// TwinCAT 3 PLC project modulx
// ProgramVersion: 3.1.0.8
// libraries:
//   Tc2_Standard, * (Beckhoff Automation GmbH)
//   Tc2_System, * (Beckhoff Automation GmbH)
//   Tc3_Interfaces, * (Beckhoff Automation GmbH)
//   Tc3_Module, * (Beckhoff Automation GmbH)
//   Tc2_MC2,3.3.5.0,Beckhoff Automation GmbH
//   Tc2_TcpIp,3.3.2.0,Beckhoff Automation GmbH
//   Tc2_Utilities,3.3.7.0,Beckhoff Automation GmbH
// project tree:
//   DataTypes/ eMainState.TcDUT, eSubState.TcDUT
//   DUTs/ArrayInterFaceDUT/DUTs/Module Interface/ DUT_MODULE_INTERFACE.TcDUT
//   DUTs/ArrayInterFaceDUT/DUTs/Module Interface/Input/ DUT_MODULE_INTERFACE_INPUT.TcDUT, DUT_SKILL_INPUT.TcDUT
//   DUTs/ArrayInterFaceDUT/DUTs/Module Interface/Output/ DUT_MODULE_INTERFACE_OUTPUT.TcDUT, DUT_SKILL_OUTPUT.TcDUT
//   DUTs/ DUT_SIMULATION.TcDUT
//   DUTs/industrialPhysics/ MNG_APPLICATION_INPUTS_32BIT.TcDUT, MNG_APPLICATION_OUTPUTS_32BIT.TcDUT, MNG_DataArray.TcDUT, MNG_DatagramHeader.TcDUT, MNG_DatagramType.TcDUT, MNG_POSE6.TcDUT, MNG_RawDatagram.TcDUT, MNG_TRAFO.TcDUT, VEC3.TcDUT
//   DUTs/Server DUTs/ DUT_MODE.TcDUT, DUT_PARAMETER_INPUT.TcDUT, DUT_PARAMETER_OUTPUT.TcDUT, DUT_SERVER_MODULE_INTERFACE.TcDUT, DUT_SERVER_MODULE_INTERFACE_INPUT.TcDUT, DUT_SERVER_MODULE_INTERFACE_OUTPUT.TcDUT, DUT_SERVER_PARAMETERINPUTARRAY.TcDUT, DUT_SERVER_PARAMETEROUTPUTARRAY.TcDUT, DUT_SERVER_SKILLINPUTARRAY.TcDUT, DUT_SERVER_SKILLOUTPUTARRAY.TcDUT, DUT_SERVER_SKILL_INPUT.TcDUT, DUT_SERVER_SKILL_OUTPUT.TcDUT, DUT_SERVER_STATEVALUEARRAY.TcDUT, DUT_SIMU_SKILLSTATE.TcDUT, DUT_STATEVALUES.TcDUT
//   GVLs/ GVL.TcGVL, MI5.TcGVL, MNG_GLOBALS.TcGVL, OPCConstants.TcGVL
//   / PlcTask.TcTTO, SimuTask.TcTTO
//   POUs/ FB_FAKE_MODULE.TcPOU, FB_Translate.TcPOU, MAIN.TcPOU
//   POUs/industrialPhysics/ FB_LogFifo.TcPOU, MAIN_simu.TcPOU, MNG_SIMULATION.TcPOU, MNG_UPDATEIOS.TcPOU
// real-time tasks:
//   TASK PlcTask: cycle T#10ms, priority 20, ADS port 350
//   TASK SimuTask: cycle T#10ms, priority 21, ADS port 351
// motion (NC):
//   TASK NC-Task 1 SAF: cycle T#2ms, priority 4, ADS port 501
//   TASK NC-Task 1 SVB: cycle T#10ms, priority 8, ADS port 511

CONFIGURATION modulx
    RESOURCE PLC ON TwinCAT3
        TASK PlcTask(INTERVAL := T#10ms, PRIORITY := 20);
        TASK SimuTask(INTERVAL := T#10ms, PRIORITY := 21);
        PROGRAM MAIN WITH PlcTask : MAIN;
        PROGRAM MAIN_simu WITH SimuTask : MAIN_simu;
    END_RESOURCE
END_CONFIGURATION

// ---- DataTypes/eMainState.TcDUT
TYPE eMainState :
(
	init		:= 0,
	ready		:= 10,
	output		:= 20,
	separation	:= 30,
	refill		:= 40
);
END_TYPE

// ---- DataTypes/eSubState.TcDUT
TYPE eSubState :
(
	step0 := 0,
	step1 := 1,
	step2 := 2,
	step3 := 3,
	step4 := 4,
	step5 := 5,
	step6 := 6,
	step7 := 7,
	step8 := 8,
	step9 := 9,
	step10 := 10,
	step11 := 11,
	step12 := 12,
	step13 := 13,
	step14 := 14,
	step15 := 15
);
END_TYPE

// ---- DUTs/ArrayInterFaceDUT/DUTs/Module Interface/DUT_MODULE_INTERFACE.TcDUT
/// MODULE INTERFACE INPUT AND OUTPUT 
TYPE DUT_MODULE_INTERFACE :
STRUCT
	///Information that the module reads
	Input: DUT_MODULE_INTERFACE_INPUT;
	///Information that the module write
	Output: DUT_MODULE_INTERFACE_OUTPUT;
END_STRUCT
END_TYPE

// ---- DUTs/ArrayInterFaceDUT/DUTs/Module Interface/Input/DUT_MODULE_INTERFACE_INPUT.TcDUT
TYPE DUT_MODULE_INTERFACE_INPUT :
STRUCT
	///Mode to run (init,auto,manual,..)
	Mode: DUT_MODE;
	///check if the modules is alive
	ConnectionTestInput: BOOL;
	///Modules get their position
	PositionInput: LREAL;
	///Update data= TRUE, No updatedata=FALSE
	Watchbit: BOOL;
	///Emergency stop
	EmergencyStop: BOOL;
	///Range of INPUT skills
	SkillInput: ARRAY[0..SkillCnt] OF DUT_SKILL_INPUT;
END_STRUCT
END_TYPE

// ---- DUTs/ArrayInterFaceDUT/DUTs/Module Interface/Input/DUT_SKILL_INPUT.TcDUT
TYPE DUT_SKILL_INPUT :
STRUCT
	///Range of parameters
	ParameterInput: ARRAY[0..ParameterCnt] OF DUT_PARAMETER_INPUT;
	///Start process
	Execute: BOOL;
END_STRUCT
END_TYPE

// ---- DUTs/ArrayInterFaceDUT/DUTs/Module Interface/Output/DUT_MODULE_INTERFACE_OUTPUT.TcDUT
TYPE DUT_MODULE_INTERFACE_OUTPUT :
STRUCT
	///Free to use = TRUE, busy to use =FALSE
	Dummy: BOOL := TRUE;
	///Individual name of the module
	Name: STRING(80);
	///Identification number of module
	ID: UINT;
	///IP address
	IP: STRING(80);
	///Show if the module is in Standby or not
	Idle: BOOL;
	///Show if the module is connected
	Connected: BOOL;
	///Feedback with conection test input
	ConnectionTestOutput: BOOL;
	///Show if the system has error when=TRUE
	Error: BOOL;
	///Identification number of the error
	ErrorID: UINT;
	///Description of the error
	ErrorDescription: STRING(80);
	///Description of the current task
	CurrentTaskDescription: STRING(80);
	///actual position of the modules, calculated by the module itself
	PositionOutput: LREAL;
	///Position of the sensor
	PositionSensor: BOOL;
	///Range of OUTPUT skills
	SkillOutput: ARRAY[0..SkillCnt] OF DUT_SKILL_OUTPUT;
	///Range of state values
	StateValue: ARRAY[0..StateCnt] OF DUT_STATEVALUES;
END_STRUCT
END_TYPE

// ---- DUTs/ArrayInterFaceDUT/DUTs/Module Interface/Output/DUT_SKILL_OUTPUT.TcDUT
TYPE DUT_SKILL_OUTPUT :
STRUCT
	///Free to use = TRUE, busy to use =FALSE
	Dummy: BOOL := TRUE;
	///Identification number of skill
	ID: UINT;
	///indentfication name of skill
	Name: STRING(80);
	///Skill activated
	Activated: BOOL;
	///Ready to do skill
	Ready: BOOL;
	///Skill in process
	Busy: BOOL;
	///Skill finish
	Done: BOOL;
	///Error in system
	Error: BOOL;
	///Range of parameters
	ParameterOutput: ARRAY[0..ParameterCnt] OF DUT_PARAMETER_OUTPUT;
END_STRUCT
END_TYPE

// ---- DUTs/DUT_SIMULATION.TcDUT
TYPE DUT_SIMULATION :
STRUCT
XPosition0 : LREAL;
XPosition1 : lreal;
XPosition2 : lreal;
XPosition3 : lreal;
XPosition4 : lreal;
XPosition5 : lreal;
XPosition6 : lreal;
XPosition7 : lreal;
XPosition8 : lreal;
XPosition9 : lreal;
XPosition10 :LREAL;

Cocktail			: DUT_SIMU_SKILLSTATE;
Cookie				: DUT_SIMU_SKILLSTATE;
Topping_Beckhoff	: DUT_SIMU_SKILLSTATE;
Topping_Bosch		: DUT_SIMU_SKILLSTATE;

END_STRUCT
END_TYPE

// ---- DUTs/industrialPhysics/MNG_APPLICATION_INPUTS_32BIT.TcDUT

TYPE MNG_APPLICATION_INPUTS_32BIT :
STRUCT
    NumSignals                     : INT     := 1         ;
    init_sensor_module_x_00_IR : BOOL    := 0; (* Physics://physics/Modulel_X/init_sensor_module_x?IR *)
END_STRUCT
END_TYPE

// ---- DUTs/industrialPhysics/MNG_APPLICATION_OUTPUTS_32BIT.TcDUT

TYPE MNG_APPLICATION_OUTPUTS_32BIT :
STRUCT
    NumSignals                     : INT     := 18        ;
    MotorX_00_par1 : BOOL    := 0; (* Physics://physics/Modulel_X/MotorX?par1 *)
    MotorX_00_par2 : BOOL    := 0; (* Physics://physics/Modulel_X/MotorX?par2 *)
    Keksmodul_00_ACT_POS02 : REAL    := 0.0; (* Physics://physics/Keksmodul?KinActual *)
    Toppingmodul_Bosch_00_ACT_POS02 : REAL    := 0.0; (* Physics://physics/Toppingmodul_Bosch?KinActual *)
    Toppingmodul_Beckhoff_00_ACT_POS02 : REAL    := 0.0; (* Physics://physics/Toppingmodul_Beckhoff?KinActual *)
    DosierModul_00_ACT_POS02 : REAL    := 0.0; (* Physics://physics/DosierModul?KinActual *)
    status_00_on102 : BOOL    := 0; (* Physics://physics/Keksmodul/status_plate/status?on1 *)
    status_00_on202 : BOOL    := 0; (* Physics://physics/Keksmodul/status_plate/status?on2 *)
    status_00_on302 : BOOL    := 0; (* Physics://physics/Keksmodul/status_plate/status?on3 *)
    status_00_on103 : BOOL    := 0; (* /physics/Toppingmodul_Bosch/status_plate/status?on1 *)
    status_00_on203 : BOOL    := 0; (* /physics/Toppingmodul_Bosch/status_plate/status?on2 *)
    status_00_on303 : BOOL    := 0; (* /physics/Toppingmodul_Bosch/status_plate/status?on3 *)
    status_00_on104 : BOOL    := 0; (* ysics/Toppingmodul_Beckhoff/status_plate/status?on1 *)
    status_00_on204 : BOOL    := 0; (* ysics/Toppingmodul_Beckhoff/status_plate/status?on2 *)
    status_00_on304 : BOOL    := 0; (* ysics/Toppingmodul_Beckhoff/status_plate/status?on3 *)
    status_00_on105 : BOOL    := 0; (* ysics://physics/DosierModul/status_plate/status?on1 *)
    status_00_on205 : BOOL    := 0; (* ysics://physics/DosierModul/status_plate/status?on2 *)
    status_00_on305 : BOOL    := 0; (* ysics://physics/DosierModul/status_plate/status?on3 *)
END_STRUCT
END_TYPE

// ---- DUTs/industrialPhysics/MNG_DataArray.TcDUT
TYPE MNG_DataArray : ARRAY[1..MNG_BUFFER_SIZE] OF DWORD; (* user data of max. length *)
END_TYPE

// ---- DUTs/industrialPhysics/MNG_DatagramHeader.TcDUT
TYPE MNG_DatagramHeader :(* datagram header (4 byte aligned) *)
STRUCT
	(* Time when datagram has been created *)
	Counter 	: DWORD;
	(* Time when datagram has been sent *)
	SentTime 		: DWORD;
	(* Type of the datagram *)
	DatagramType 	: DWORD := MNG_UnknownDatagram;
	(* Byte count in the payload *)
	ByteCount 		: DWORD := 0;
END_STRUCT
END_TYPE

// ---- DUTs/industrialPhysics/MNG_DatagramType.TcDUT
TYPE MNG_DatagramType :
(
	(*Dead man datagram signalizing peer is alive *)
	MNG_DeadManDatagram := 0,
	(*Time tick synchonisation *)
	MNG_TimeTick,
	(*Time tick synchonisation *)
	MNG_TimeTickRequest,
	(*Initialization of the connection *)
	MNG_InitConnection,
	(*Reset simulation *)
	MNG_ResetSimulation,
	(*Rewind simulation *)
	MNG_RewindSimulation,
	(*Start simulation *)
	MNG_StartSimulation,
	(*Stop simulation *)
	MNG_StopSimulation,
	(*IO Config datagram *)
	MNG_IOConfig,
	(*Complete Raw IO Image *)
	MNG_RawIOImage,
	(*Complete Raw 32 Bit IO Image *)
	MNG_Raw32BitImage,
	(*Delta IO, only ios that have changed *)
	(* IODelta, *)
	(*Text datagram *)
	MNG_TextDatagram,
	(*Unknown Datagram (future updates of peer, not supported by this side) *)
	MNG_UnknownDatagram
);
END_TYPE

// ---- DUTs/industrialPhysics/MNG_POSE6.TcDUT
TYPE MNG_POSE6 :(* position and orientation as an euler based pose *)
STRUCT
	x, y, z, a, b, c : REAL;
END_STRUCT
END_TYPE

// ---- DUTs/industrialPhysics/MNG_RawDatagram.TcDUT
TYPE MNG_RawDatagram :(* binary TCP/IP datagram (4 byte aligned) *)
STRUCT
	Header	:  MNG_DatagramHeader;(* datagram header *)
	Payload	:  MNG_DataARRAY;
END_STRUCT
END_TYPE

// ---- DUTs/industrialPhysics/MNG_TRAFO.TcDUT
TYPE MNG_TRAFO :(* position and orientation as a 4x4 matrix *)
STRUCT
	baseX : VEC3; 
	fill0 : REAL;
	baseY : VEC3; 
	fill1 : REAL;
	baseZ : VEC3; 
	fill2 : REAL;
	origin : VEC3;
	fill3 : REAL;
END_STRUCT
END_TYPE

// ---- DUTs/industrialPhysics/VEC3.TcDUT
TYPE VEC3 :(* 3d position *)
STRUCT
	x, y, z : REAL;
END_STRUCT
END_TYPE

// ---- DUTs/Server DUTs/DUT_MODE.TcDUT
/// MODE to run (inside of MODULE_INTERFACE_INPUT)
TYPE DUT_MODE :
(
	///Initialitzation number mode
	Init := 0,
	///Automatic number mode
	Auto := 1,
	///Manual number mode
	Manual := 2,
	Reset := 3
);
END_TYPE

// ---- DUTs/Server DUTs/DUT_PARAMETER_INPUT.TcDUT
TYPE DUT_PARAMETER_INPUT :
STRUCT
	///Value of the parameter 
	Value: LREAL;
	///Possibility to a string value depending on the parameter
	StringValue: STRING(80);
END_STRUCT
END_TYPE

// ---- DUTs/Server DUTs/DUT_PARAMETER_OUTPUT.TcDUT
TYPE DUT_PARAMETER_OUTPUT :
STRUCT
	///Free to use = TRUE, busy to use =FALSE
	Dummy: BOOL := TRUE;
	///ID of the parameter
	ID: UINT;
	///Name of the parameter
	Name: STRING(80);
	///Unit of the parameter
	Unit: STRING(80);
	///Optional parameter
	Required: BOOL;
	///Default parameter to work
	Default: LREAL;
	///Minimum value of the parameter
	MinValue: LREAL;
	///Maximum value of the parameter
	MaxValue: LREAL;
END_STRUCT
END_TYPE

// ---- DUTs/Server DUTs/DUT_SERVER_MODULE_INTERFACE.TcDUT
/// MODULE INTERFACE INPUT AND OUTPUT 
TYPE DUT_SERVER_MODULE_INTERFACE :
STRUCT
	///Information that the module reads
	Input: DUT_SERVER_MODULE_INTERFACE_INPUT;
	///Information that the module write
	Output: DUT_SERVER_MODULE_INTERFACE_OUTPUT;
END_STRUCT
END_TYPE

// ---- DUTs/Server DUTs/DUT_SERVER_MODULE_INTERFACE_INPUT.TcDUT
TYPE DUT_SERVER_MODULE_INTERFACE_INPUT :
STRUCT
	///Mode to run (init,auto,manual,..)
	Mode: INT;//DUT_MODE;
	///check if the modules is alive
	ConnectionTestInput: BOOL;
	///Modules get their position
	PositionInput: LREAL;
	///Update data= TRUE, No updatedata=FALSE
	Watchbit: BOOL;
	///Emergency stop
	EmergencyStop: BOOL;
	///Range of INPUT skills
	SkillInput: DUT_SERVER_SKILLINPUTARRAY;
END_STRUCT
END_TYPE

// ---- DUTs/Server DUTs/DUT_SERVER_MODULE_INTERFACE_OUTPUT.TcDUT
TYPE DUT_SERVER_MODULE_INTERFACE_OUTPUT :
STRUCT
	///Free to use = TRUE, busy to use =FALSE
	Dummy: BOOL := TRUE;
	///Individual name of the module
	Name: STRING(80);
	///Identification number of module
	ID: UINT;
	///IP address
	IP: STRING(80);
	///Show if the module is in Standby or not
	Idle: BOOL;
	///Show if the module is connected
	Connected: BOOL;
	///Feedback with conection test input
	ConnectionTestOutput: BOOL;
	///Show if the system has error when=TRUE
	Error: BOOL;
	///Identification number of the error
	ErrorID: UINT;
	///Description of the error
	ErrorDescription: STRING(80);
	///Description of the current task
	CurrentTaskDescription: STRING(80);
	///Position of the output
	PositionOutput: LREAL;
	/// Bool value of the Sensor
	PositionSensor: BOOL;
	///Range of OUTPUT skills
	SkillOutput: DUT_SERVER_SKILLOUTPUTARRAY;
	///Range of state values
	StateValue: DUT_SERVER_STATEVALUEARRAY;
END_STRUCT
END_TYPE

// ---- DUTs/Server DUTs/DUT_SERVER_PARAMETERINPUTARRAY.TcDUT
TYPE DUT_SERVER_PARAMETERINPUTARRAY :
STRUCT
	ParameterInput0: DUT_PARAMETER_INPUT;
	ParameterInput1: DUT_PARAMETER_INPUT;
	ParameterInput2: DUT_PARAMETER_INPUT;
	ParameterInput3: DUT_PARAMETER_INPUT;
	ParameterInput4: DUT_PARAMETER_INPUT;
	ParameterInput5: DUT_PARAMETER_INPUT;
END_STRUCT
END_TYPE

// ---- DUTs/Server DUTs/DUT_SERVER_PARAMETEROUTPUTARRAY.TcDUT
TYPE DUT_SERVER_PARAMETEROUTPUTARRAY :
STRUCT
	ParameterOutput0: DUT_PARAMETER_OUTPUT;
	ParameterOutput1: DUT_PARAMETER_OUTPUT;
	ParameterOutput2: DUT_PARAMETER_OUTPUT;
	ParameterOutput3: DUT_PARAMETER_OUTPUT;
	ParameterOutput4: DUT_PARAMETER_OUTPUT;
	ParameterOutput5: DUT_PARAMETER_OUTPUT;
END_STRUCT
END_TYPE

// ---- DUTs/Server DUTs/DUT_SERVER_SKILLINPUTARRAY.TcDUT
TYPE DUT_SERVER_SKILLINPUTARRAY :
STRUCT
	SkillInput0: DUT_SERVER_SKILL_INPUT;
	SkillInput1: DUT_SERVER_SKILL_INPUT;
	SkillInput2: DUT_SERVER_SKILL_INPUT;
	SkillInput3: DUT_SERVER_SKILL_INPUT;
	SkillInput4: DUT_SERVER_SKILL_INPUT;
	SkillInput5: DUT_SERVER_SKILL_INPUT;
	SkillInput6: DUT_SERVER_SKILL_INPUT;
	SkillInput7: DUT_SERVER_SKILL_INPUT;
	SkillInput8: DUT_SERVER_SKILL_INPUT;
	SkillInput9: DUT_SERVER_SKILL_INPUT;
	SkillInput10: DUT_SERVER_SKILL_INPUT;
	SkillInput11: DUT_SERVER_SKILL_INPUT;
	SkillInput12: DUT_SERVER_SKILL_INPUT;
	SkillInput13: DUT_SERVER_SKILL_INPUT;
	SkillInput14: DUT_SERVER_SKILL_INPUT;
	SkillInput15: DUT_SERVER_SKILL_INPUT;
END_STRUCT
END_TYPE

// ---- DUTs/Server DUTs/DUT_SERVER_SKILLOUTPUTARRAY.TcDUT
TYPE DUT_SERVER_SKILLOUTPUTARRAY :
STRUCT
	SkillOutput0: DUT_SERVER_SKILL_OUTPUT;
	SkillOutput1: DUT_SERVER_SKILL_OUTPUT;
	SkillOutput2: DUT_SERVER_SKILL_OUTPUT;
	SkillOutput3: DUT_SERVER_SKILL_OUTPUT;
	SkillOutput4: DUT_SERVER_SKILL_OUTPUT;
	SkillOutput5: DUT_SERVER_SKILL_OUTPUT;
	SkillOutput6: DUT_SERVER_SKILL_OUTPUT;
	SkillOutput7: DUT_SERVER_SKILL_OUTPUT;
	SkillOutput8: DUT_SERVER_SKILL_OUTPUT;
	SkillOutput9: DUT_SERVER_SKILL_OUTPUT;
	SkillOutput10: DUT_SERVER_SKILL_OUTPUT;
	SkillOutput11: DUT_SERVER_SKILL_OUTPUT;
	SkillOutput12: DUT_SERVER_SKILL_OUTPUT;
	SkillOutput13: DUT_SERVER_SKILL_OUTPUT;
	SkillOutput14: DUT_SERVER_SKILL_OUTPUT;
	SkillOutput15: DUT_SERVER_SKILL_OUTPUT;
END_STRUCT
END_TYPE

// ---- DUTs/Server DUTs/DUT_SERVER_SKILL_INPUT.TcDUT
TYPE DUT_SERVER_SKILL_INPUT :
STRUCT
	///Range of parameters
	ParameterInput: DUT_SERVER_PARAMETERINPUTARRAY;
	///Start process
	Execute: BOOL;
END_STRUCT
END_TYPE

// ---- DUTs/Server DUTs/DUT_SERVER_SKILL_OUTPUT.TcDUT
TYPE DUT_SERVER_SKILL_OUTPUT :
STRUCT
	///Free to use = TRUE, busy to use =FALSE
	Dummy: BOOL := TRUE;
	///Identification number of skill
	ID: UINT;
	///indentfication name of skill
	Name: STRING(80);
	///Skill activated
	Activated: BOOL;
	///Ready to do skill
	Ready: BOOL;
	///Skill in process
	Busy: BOOL;
	///Skill finish
	Done: BOOL;
	///Error in system
	Error: BOOL;
	///Range of parameters
	ParameterOutput: DUT_SERVER_PARAMETEROUTPUTARRAY;
END_STRUCT
END_TYPE

// ---- DUTs/Server DUTs/DUT_SERVER_STATEVALUEARRAY.TcDUT
TYPE DUT_SERVER_STATEVALUEARRAY :
STRUCT
	StateValue0: DUT_STATEVALUES;
	StateValue1: DUT_STATEVALUES;
	StateValue2: DUT_STATEVALUES;
	StateValue3: DUT_STATEVALUES;
	StateValue4: DUT_STATEVALUES;
	StateValue5: DUT_STATEVALUES;
	StateValue6: DUT_STATEVALUES;
	StateValue7: DUT_STATEVALUES;
	StateValue8: DUT_STATEVALUES;
	StateValue9: DUT_STATEVALUES;
	StateValue10: DUT_STATEVALUES;
END_STRUCT
END_TYPE

// ---- DUTs/Server DUTs/DUT_SIMU_SKILLSTATE.TcDUT
TYPE DUT_SIMU_SKILLSTATE :
STRUCT
	
Ready 	:BOOL;
Busy	:BOOL;
Error	:BOOL;

END_STRUCT
END_TYPE

// ---- DUTs/Server DUTs/DUT_STATEVALUES.TcDUT
TYPE DUT_STATEVALUES :
STRUCT
	///Free to use = TRUE, busy to use =FALSE
	Dummy: BOOL := TRUE;
	///Value of the State
	Value: LREAL;
	///Name of the state
	Name: STRING(80);
	///Description of the state
	Description: STRING(80);
	///Unit of the state ()
	Unit: STRING(80);
END_STRUCT
END_TYPE

// ---- GVLs/GVL.TcGVL
VAR_GLOBAL
	pi : REAL := 3.14159;
																
	//<<Input Variables>>//
	iOrder 			AT%I*	: BOOL; 				// is there a order to separate cookies? --> from database
	iDiskAtStorage 	AT%I*	: BOOL; 				// is the gap of the disk at the storage? --> from hall sensor
	iDiskAtRamp 	AT%I*	: BOOL;					// is the gap of the disk at the ramp? --> from hall sensor
	iCookieInOutput	AT%I*	: BOOL;					// is the cookie in the ouput (on the clamp)? --> from light barrier sensor
	iStorageLevel 	AT%I*	: INT;					// number of remaining cookies in the storage --> from distance sensor
	iClearence		AT%I*	: BOOL;					// did the user clear the refilling/maintenance process --> from HMI
	
	//<<Output Variables>>//
	oTurnDiskLeft	AT%Q*	: BOOL := FALSE;		// turn disk anti-clockwise/left 
										 			//@TODO: later as a function with choosable fastVel/acceleration/...
	oTurnDiskRight	AT%Q*	: BOOL := FALSE;		// turn disk anti-clockwise/left 
										 			//@TODO: later as a function with choosable fastVel/acceleration/...							
	//oStorageEmpty	AT%Q*	: BOOL := FALSE;		// ???? message to HMI about cookie storage
	oHMIMessage		AT%Q*	: STRING :='';			//message to HMI depending on current state
	
	//<<Internal Variables>>//
	mainState 				: eMainState		:= eMainState.init;
	subState				: eSubState 		:= eSubState.step0;	
	
	axis	 				: AXIS_REF;
	fastVel					: INT	:= 40;
	slowVel					: INT	:= 20;
	
	
	
	
	//<<For Visualization>>//
	init_					: BOOL := FALSE;
	ready_					: BOOL := FALSE;
	output_					: BOOL := FALSE;
	separation_				: BOOL := FALSE;
	refill_					: BOOL := FALSE;
	
	offset					: LREAL;
	infinitsimu				: BOOL;
	infinitsimu2			: BOOL;	
	sensorPosition			: LREAL;
	
	init_sensor_x			: BOOL;
	lamp1				: BOOL;
	lamp2				: BOOL;	
END_VAR

// ---- GVLs/MI5.TcGVL
VAR_GLOBAL
	//<<OPC-UA Module Interface>>//
	{attribute 'OPC.UA.DA' := '1'}
	Module1202 : DUT_SERVER_MODULE_INTERFACE;
	{attribute 'OPC.UA.DA' := '1'}
	Module2501 : DUT_SERVER_MODULE_INTERFACE;
	{attribute 'OPC.UA.DA' := '1'}
	Module2601 : DUT_SERVER_MODULE_INTERFACE;
	{attribute 'OPC.UA.DA' := '1'}
	Simulation: DUT_SIMULATION;
	{attribute 'OPC.UA.DA' := '1'}	
	ResetProcessTool 	: BOOL;
	
	// INTERN MODULE INTERFACE
	InternalModule	: DUT_MODULE_INTERFACE;
END_VAR

// ---- GVLs/MNG_GLOBALS.TcGVL

VAR_GLOBAL CONSTANT
	PLCPRJ_MAX_CONNECTIONS					: UDINT 	:= 5;   (* Max. number of server<->client connections *)
	PLCPRJ_SERVER_RESPONSE_TIMEOUT			: TIME 	:= T#10s;
	PLCPRJ_CLIENT_SEND_CYCLE_TIME			: TIME 	:= T#1ms;

	PLCPRJ_RECEIVER_POLLING_CYCLE_TIME		: TIME 	:= T#1ms;
	PLCPRJ_BUFFER_SIZE						: UDINT	:= 10000;   (* Max. internal fifo/receiver buffer size *)

	(* Some project specific error codes *)
	PLCPRJ_ERROR_RECEIVE_BUFFER_OVERFLOW	: UDINT := 16#8101; (* receive fifo/buffer overflow*)
	PLCPRJ_ERROR_SEND_BUFFER_OVERFLOW		: UDINT := 16#8102;	(* send fifo/buffer overflow *)
	PLCPRJ_ERROR_RESPONSE_TIMEOUT			: UDINT := 16#8103;	(* receive timeout error *)
	
	

	PLCPRJ_ERROR_INVALID_FRAME_FORMAT		: UDINT := 16#8104;	(* invalid frame format/data *)
	PLCPRJ_ERROR_INVALID_IO_FORMAT_RECEIVED : UDINT := 16#8105;	(* invalid io format/data *)
	PLCPRJ_ERROR_INTERNAL					: UDINT := 16#8105; (* internal error *)
	PLCPRJ_ERROR_RX_DATA_INCONSISTENT		: UDINT := 16#8106; (* rx data inconsistent *)
	
	PLCPRJ_ERROR_RECEIVE_TIMEOUT			: UDINT := 16#8107;
	PLCPRJ_ERROR_SENDFIFO_OVERFLOW			: UDINT := 16#8108; (* send fifo overflow error *)
	PLCPRJ_ERROR_RECFIFO_OVERFLOW			: UDINT := 16#8109; (* receive fifo overflow error *)
	
    MNG_BUFFER_SIZE						: DWORD := 32768;   (* Bytes: 131072; Max 128 KB of datagram payload data*)
	MNG_DatagramsFIFO_Size					: DWORD := 10;      (* Max 10 datagrams buffered before loss occurs *)
	MNG_EmptyDatagramHeader					: MNG_DatagramHeader;
	MNG_Application_NumInputs				: DWORD := 4;
	MNG_Application_NumOutputs				: DWORD := 4;

        (* PI should be defined by the system *)
        (* PI      : LREAL := 3.1415926535897932384626433832795; *)
        DEG2RAD : LREAL := 0.017453292519943295769236907684886;
        RAD2DEG : LREAL := 57.295779513082320876798154814105;
END_VAR

VAR_GLOBAL
        MNG_TIMESTAMP                                           : LREAL := 0;
END_VAR

// ---- GVLs/OPCConstants.TcGVL
VAR_GLOBAL CONSTANT
	///Maximum number of skillparameters
	ParameterCnt: INT := 5;
	///Maximum number of skills per Module
	SkillCnt: INT := 15;
	///Maximum number of Statevalues of one Module
	StateCnt: INT := 10;
	///Maximum number of modules
	ModuleCnt: INT := 10;
	///Maximum number of Tasks in Production List
	TaskCnt: INT := 30;
	///Maximum number  of offered recipes
	OfferCnt: INT := 5;
	///Maximum number of Orders in Queue
	OrderCnt: INT := 5;
	///Number of user set parameters per recipe
	UserParameterCnt: INT := 5;
	///Number of skills per task
	TaskSkillCnt: INT := 50;
END_VAR

// ---- POUs/MAIN.TcPOU
PROGRAM MAIN
VAR


	
	fbTranslate		: FB_TRANSLATE;
	fbFakeModule	: FB_FAKE_MODULE;
	fbi_Timer: TOF;
END_VAR


//für dieses modul muss Module1102 (ausgang von fbTranslate) noch auf den richtigen modulausgang geändert werden und in den GVLs eine Variable vom Typ DUT_Module_Interface (mit arrays) und dem namen InternalModule hinzugefügt werden
// FAKE MODUL:	
fbFakeModule.SKILLID[0] := 1337;

fbFakeModule(INPUT:=InternalModule.Input, OUTPUT => InternalModule.Output,  Execute := TRUE );
fbTranslate(ArrayModule := InternalModule, ServerModule := Module1202);
fbi_Timer();

// sensorhigh delay erzeugen/verlängern
IF GVL.init_sensor_x THEN
	Module1202.Output.PositionSensor := TRUE;
	
	fbi_Timer(IN := TRUE,PT := T#400MS);
	fbi_Timer(IN := FALSE,PT := T#400MS);	
ELSE
	Module1202.Output.PositionSensor := fbi_Timer.Q;
END_IF

Module2501.Output.PositionOutput := 1345.0;
Module2601.Output.PositionOutput := 165.0;

END_PROGRAM

// ---- POUs/FB_Translate.TcPOU
FUNCTION_BLOCK FB_Translate
VAR_INPUT
	execute : BOOL := TRUE;
END_VAR
VAR_OUTPUT
END_VAR
VAR

 
END_VAR
VAR_IN_OUT
	ArrayModule	: DUT_MODULE_INTERFACE;
	ServerModule: DUT_SERVER_MODULE_INTERFACE;
END_VAR

IF execute THEN
	ArrayModule.Input.Mode := ServerModule.Input.Mode;
ArrayModule.Input.ConnectionTestInput := ServerModule.Input.ConnectionTestInput;
ArrayModule.Input.PositionInput := ServerModule.Input.PositionInput;
ArrayModule.Input.Watchbit := ServerModule.Input.Watchbit;
ArrayModule.Input.EmergencyStop := ServerModule.Input.EmergencyStop;
ServerModule.Output.Dummy := ArrayModule.Output.Dummy;
ServerModule.Output.Name := ArrayModule.Output.Name;
ServerModule.Output.ID := ArrayModule.Output.ID;
ServerModule.Output.IP := ArrayModule.Output.IP;
ServerModule.Output.Idle := ArrayModule.Output.Idle;
ServerModule.Output.Connected := ArrayModule.Output.Connected;
ServerModule.Output.Error := ArrayModule.Output.Error;
ServerModule.Output.ErrorID := ArrayModule.Output.ErrorID;
ServerModule.Output.ErrorDescription := ArrayModule.Output.ErrorDescription;
ServerModule.Output.CurrentTaskDescription := ArrayModule.Output.CurrentTaskDescription;
ServerModule.Output.PositionSensor := ArrayModule.Output.PositionSensor;
ServerModule.Output.ConnectionTestOutput := ArrayModule.Output.ConnectionTestOutput;
ServerModule.Output.PositionOutput := ArrayModule.Output.PositionOutput;
ArrayModule.Input.SkillInput[0].Execute := ServerModule.Input.SkillInput.SkillInput0.Execute;
ServerModule.Output.SkillOutput.SkillOutput0.Dummy := ArrayModule.Output.SkillOutput[0].Dummy;
ServerModule.Output.SkillOutput.SkillOutput0.ID := ArrayModule.Output.SkillOutput[0].ID;
ServerModule.Output.SkillOutput.SkillOutput0.Name := ArrayModule.Output.SkillOutput[0].Name;
ServerModule.Output.SkillOutput.SkillOutput0.Activated := ArrayModule.Output.SkillOutput[0].Activated;
ServerModule.Output.SkillOutput.SkillOutput0.Ready := ArrayModule.Output.SkillOutput[0].Ready;
ServerModule.Output.SkillOutput.SkillOutput0.Busy := ArrayModule.Output.SkillOutput[0].Busy;
ServerModule.Output.SkillOutput.SkillOutput0.Done := ArrayModule.Output.SkillOutput[0].Done;
ServerModule.Output.SkillOutput.SkillOutput0.Error := ArrayModule.Output.SkillOutput[0].Error;
ServerModule.Output.Statevalue.Statevalue0 := ArrayModule.Output.Statevalue[0];
ServerModule.Output.Statevalue.Statevalue1 := ArrayModule.Output.Statevalue[1];
ServerModule.Output.Statevalue.Statevalue2 := ArrayModule.Output.Statevalue[2];
ServerModule.Output.Statevalue.Statevalue3 := ArrayModule.Output.Statevalue[3];
ServerModule.Output.Statevalue.Statevalue4 := ArrayModule.Output.Statevalue[4];
ServerModule.Output.Statevalue.Statevalue5 := ArrayModule.Output.Statevalue[5];
ServerModule.Output.Statevalue.Statevalue6 := ArrayModule.Output.Statevalue[6];
ServerModule.Output.Statevalue.Statevalue7 := ArrayModule.Output.Statevalue[7];
ServerModule.Output.Statevalue.Statevalue8 := ArrayModule.Output.Statevalue[8];
ServerModule.Output.Statevalue.Statevalue9 := ArrayModule.Output.Statevalue[9];
ServerModule.Output.Statevalue.Statevalue10 := ArrayModule.Output.Statevalue[10];
ArrayModule.Input.SkillInput[0].ParameterInput[0] := ServerModule.Input.SkillInput.SkillInput0.ParameterInput.ParameterInput0;
ServerModule.Output.SkillOutput.SkillOutput0.ParameterOutput.ParameterOutput0 := ArrayModule.Output.SkillOutput[0].ParameterOutput[0];
ArrayModule.Input.SkillInput[0].ParameterInput[1] := ServerModule.Input.SkillInput.SkillInput0.ParameterInput.ParameterInput1;
ServerModule.Output.SkillOutput.SkillOutput0.ParameterOutput.ParameterOutput1 := ArrayModule.Output.SkillOutput[0].ParameterOutput[1];
ArrayModule.Input.SkillInput[0].ParameterInput[2] := ServerModule.Input.SkillInput.SkillInput0.ParameterInput.ParameterInput2;
ServerModule.Output.SkillOutput.SkillOutput0.ParameterOutput.ParameterOutput2 := ArrayModule.Output.SkillOutput[0].ParameterOutput[2];
ArrayModule.Input.SkillInput[0].ParameterInput[3] := ServerModule.Input.SkillInput.SkillInput0.ParameterInput.ParameterInput3;
ServerModule.Output.SkillOutput.SkillOutput0.ParameterOutput.ParameterOutput3 := ArrayModule.Output.SkillOutput[0].ParameterOutput[3];
ArrayModule.Input.SkillInput[0].ParameterInput[4] := ServerModule.Input.SkillInput.SkillInput0.ParameterInput.ParameterInput4;
ServerModule.Output.SkillOutput.SkillOutput0.ParameterOutput.ParameterOutput4 := ArrayModule.Output.SkillOutput[0].ParameterOutput[4];
ArrayModule.Input.SkillInput[0].ParameterInput[5] := ServerModule.Input.SkillInput.SkillInput0.ParameterInput.ParameterInput5;
ServerModule.Output.SkillOutput.SkillOutput0.ParameterOutput.ParameterOutput5 := ArrayModule.Output.SkillOutput[0].ParameterOutput[5];
ArrayModule.Input.SkillInput[1].Execute := ServerModule.Input.SkillInput.SkillInput1.Execute;
ServerModule.Output.SkillOutput.SkillOutput1.Dummy := ArrayModule.Output.SkillOutput[1].Dummy;
ServerModule.Output.SkillOutput.SkillOutput1.ID := ArrayModule.Output.SkillOutput[1].ID;
ServerModule.Output.SkillOutput.SkillOutput1.Name := ArrayModule.Output.SkillOutput[1].Name;
ServerModule.Output.SkillOutput.SkillOutput1.Activated := ArrayModule.Output.SkillOutput[1].Activated;
ServerModule.Output.SkillOutput.SkillOutput1.Ready := ArrayModule.Output.SkillOutput[1].Ready;
ServerModule.Output.SkillOutput.SkillOutput1.Busy := ArrayModule.Output.SkillOutput[1].Busy;
ServerModule.Output.SkillOutput.SkillOutput1.Done := ArrayModule.Output.SkillOutput[1].Done;
ServerModule.Output.SkillOutput.SkillOutput1.Error := ArrayModule.Output.SkillOutput[1].Error;
ServerModule.Output.Statevalue.Statevalue0 := ArrayModule.Output.Statevalue[0];
ServerModule.Output.Statevalue.Statevalue1 := ArrayModule.Output.Statevalue[1];
ServerModule.Output.Statevalue.Statevalue2 := ArrayModule.Output.Statevalue[2];
ServerModule.Output.Statevalue.Statevalue3 := ArrayModule.Output.Statevalue[3];
ServerModule.Output.Statevalue.Statevalue4 := ArrayModule.Output.Statevalue[4];
ServerModule.Output.Statevalue.Statevalue5 := ArrayModule.Output.Statevalue[5];
ServerModule.Output.Statevalue.Statevalue6 := ArrayModule.Output.Statevalue[6];
ServerModule.Output.Statevalue.Statevalue7 := ArrayModule.Output.Statevalue[7];
ServerModule.Output.Statevalue.Statevalue8 := ArrayModule.Output.Statevalue[8];
ServerModule.Output.Statevalue.Statevalue9 := ArrayModule.Output.Statevalue[9];
ServerModule.Output.Statevalue.Statevalue10 := ArrayModule.Output.Statevalue[10];
ArrayModule.Input.SkillInput[1].ParameterInput[0] := ServerModule.Input.SkillInput.SkillInput1.ParameterInput.ParameterInput0;
ServerModule.Output.SkillOutput.SkillOutput1.ParameterOutput.ParameterOutput0 := ArrayModule.Output.SkillOutput[1].ParameterOutput[0];
ArrayModule.Input.SkillInput[1].ParameterInput[1] := ServerModule.Input.SkillInput.SkillInput1.ParameterInput.ParameterInput1;
ServerModule.Output.SkillOutput.SkillOutput1.ParameterOutput.ParameterOutput1 := ArrayModule.Output.SkillOutput[1].ParameterOutput[1];
ArrayModule.Input.SkillInput[1].ParameterInput[2] := ServerModule.Input.SkillInput.SkillInput1.ParameterInput.ParameterInput2;
ServerModule.Output.SkillOutput.SkillOutput1.ParameterOutput.ParameterOutput2 := ArrayModule.Output.SkillOutput[1].ParameterOutput[2];
ArrayModule.Input.SkillInput[1].ParameterInput[3] := ServerModule.Input.SkillInput.SkillInput1.ParameterInput.ParameterInput3;
ServerModule.Output.SkillOutput.SkillOutput1.ParameterOutput.ParameterOutput3 := ArrayModule.Output.SkillOutput[1].ParameterOutput[3];
ArrayModule.Input.SkillInput[1].ParameterInput[4] := ServerModule.Input.SkillInput.SkillInput1.ParameterInput.ParameterInput4;
ServerModule.Output.SkillOutput.SkillOutput1.ParameterOutput.ParameterOutput4 := ArrayModule.Output.SkillOutput[1].ParameterOutput[4];
ArrayModule.Input.SkillInput[1].ParameterInput[5] := ServerModule.Input.SkillInput.SkillInput1.ParameterInput.ParameterInput5;
ServerModule.Output.SkillOutput.SkillOutput1.ParameterOutput.ParameterOutput5 := ArrayModule.Output.SkillOutput[1].ParameterOutput[5];
ArrayModule.Input.SkillInput[2].Execute := ServerModule.Input.SkillInput.SkillInput2.Execute;
ServerModule.Output.SkillOutput.SkillOutput2.Dummy := ArrayModule.Output.SkillOutput[2].Dummy;
ServerModule.Output.SkillOutput.SkillOutput2.ID := ArrayModule.Output.SkillOutput[2].ID;
ServerModule.Output.SkillOutput.SkillOutput2.Name := ArrayModule.Output.SkillOutput[2].Name;
ServerModule.Output.SkillOutput.SkillOutput2.Activated := ArrayModule.Output.SkillOutput[2].Activated;
ServerModule.Output.SkillOutput.SkillOutput2.Ready := ArrayModule.Output.SkillOutput[2].Ready;
ServerModule.Output.SkillOutput.SkillOutput2.Busy := ArrayModule.Output.SkillOutput[2].Busy;
ServerModule.Output.SkillOutput.SkillOutput2.Done := ArrayModule.Output.SkillOutput[2].Done;
ServerModule.Output.SkillOutput.SkillOutput2.Error := ArrayModule.Output.SkillOutput[2].Error;
ServerModule.Output.Statevalue.Statevalue0 := ArrayModule.Output.Statevalue[0];
ServerModule.Output.Statevalue.Statevalue1 := ArrayModule.Output.Statevalue[1];
ServerModule.Output.Statevalue.Statevalue2 := ArrayModule.Output.Statevalue[2];
ServerModule.Output.Statevalue.Statevalue3 := ArrayModule.Output.Statevalue[3];
ServerModule.Output.Statevalue.Statevalue4 := ArrayModule.Output.Statevalue[4];
ServerModule.Output.Statevalue.Statevalue5 := ArrayModule.Output.Statevalue[5];
ServerModule.Output.Statevalue.Statevalue6 := ArrayModule.Output.Statevalue[6];
ServerModule.Output.Statevalue.Statevalue7 := ArrayModule.Output.Statevalue[7];
ServerModule.Output.Statevalue.Statevalue8 := ArrayModule.Output.Statevalue[8];
ServerModule.Output.Statevalue.Statevalue9 := ArrayModule.Output.Statevalue[9];
ServerModule.Output.Statevalue.Statevalue10 := ArrayModule.Output.Statevalue[10];
ArrayModule.Input.SkillInput[2].ParameterInput[0] := ServerModule.Input.SkillInput.SkillInput2.ParameterInput.ParameterInput0;
ServerModule.Output.SkillOutput.SkillOutput2.ParameterOutput.ParameterOutput0 := ArrayModule.Output.SkillOutput[2].ParameterOutput[0];
ArrayModule.Input.SkillInput[2].ParameterInput[1] := ServerModule.Input.SkillInput.SkillInput2.ParameterInput.ParameterInput1;
ServerModule.Output.SkillOutput.SkillOutput2.ParameterOutput.ParameterOutput1 := ArrayModule.Output.SkillOutput[2].ParameterOutput[1];
ArrayModule.Input.SkillInput[2].ParameterInput[2] := ServerModule.Input.SkillInput.SkillInput2.ParameterInput.ParameterInput2;
ServerModule.Output.SkillOutput.SkillOutput2.ParameterOutput.ParameterOutput2 := ArrayModule.Output.SkillOutput[2].ParameterOutput[2];
ArrayModule.Input.SkillInput[2].ParameterInput[3] := ServerModule.Input.SkillInput.SkillInput2.ParameterInput.ParameterInput3;
ServerModule.Output.SkillOutput.SkillOutput2.ParameterOutput.ParameterOutput3 := ArrayModule.Output.SkillOutput[2].ParameterOutput[3];
ArrayModule.Input.SkillInput[2].ParameterInput[4] := ServerModule.Input.SkillInput.SkillInput2.ParameterInput.ParameterInput4;
ServerModule.Output.SkillOutput.SkillOutput2.ParameterOutput.ParameterOutput4 := ArrayModule.Output.SkillOutput[2].ParameterOutput[4];
ArrayModule.Input.SkillInput[2].ParameterInput[5] := ServerModule.Input.SkillInput.SkillInput2.ParameterInput.ParameterInput5;
ServerModule.Output.SkillOutput.SkillOutput2.ParameterOutput.ParameterOutput5 := ArrayModule.Output.SkillOutput[2].ParameterOutput[5];
ArrayModule.Input.SkillInput[3].Execute := ServerModule.Input.SkillInput.SkillInput3.Execute;
ServerModule.Output.SkillOutput.SkillOutput3.Dummy := ArrayModule.Output.SkillOutput[3].Dummy;
ServerModule.Output.SkillOutput.SkillOutput3.ID := ArrayModule.Output.SkillOutput[3].ID;
ServerModule.Output.SkillOutput.SkillOutput3.Name := ArrayModule.Output.SkillOutput[3].Name;
ServerModule.Output.SkillOutput.SkillOutput3.Activated := ArrayModule.Output.SkillOutput[3].Activated;
ServerModule.Output.SkillOutput.SkillOutput3.Ready := ArrayModule.Output.SkillOutput[3].Ready;
ServerModule.Output.SkillOutput.SkillOutput3.Busy := ArrayModule.Output.SkillOutput[3].Busy;
ServerModule.Output.SkillOutput.SkillOutput3.Done := ArrayModule.Output.SkillOutput[3].Done;
ServerModule.Output.SkillOutput.SkillOutput3.Error := ArrayModule.Output.SkillOutput[3].Error;
ServerModule.Output.Statevalue.Statevalue0 := ArrayModule.Output.Statevalue[0];
ServerModule.Output.Statevalue.Statevalue1 := ArrayModule.Output.Statevalue[1];
ServerModule.Output.Statevalue.Statevalue2 := ArrayModule.Output.Statevalue[2];
ServerModule.Output.Statevalue.Statevalue3 := ArrayModule.Output.Statevalue[3];
ServerModule.Output.Statevalue.Statevalue4 := ArrayModule.Output.Statevalue[4];
ServerModule.Output.Statevalue.Statevalue5 := ArrayModule.Output.Statevalue[5];
ServerModule.Output.Statevalue.Statevalue6 := ArrayModule.Output.Statevalue[6];
ServerModule.Output.Statevalue.Statevalue7 := ArrayModule.Output.Statevalue[7];
ServerModule.Output.Statevalue.Statevalue8 := ArrayModule.Output.Statevalue[8];
ServerModule.Output.Statevalue.Statevalue9 := ArrayModule.Output.Statevalue[9];
ServerModule.Output.Statevalue.Statevalue10 := ArrayModule.Output.Statevalue[10];
ArrayModule.Input.SkillInput[3].ParameterInput[0] := ServerModule.Input.SkillInput.SkillInput3.ParameterInput.ParameterInput0;
ServerModule.Output.SkillOutput.SkillOutput3.ParameterOutput.ParameterOutput0 := ArrayModule.Output.SkillOutput[3].ParameterOutput[0];
ArrayModule.Input.SkillInput[3].ParameterInput[1] := ServerModule.Input.SkillInput.SkillInput3.ParameterInput.ParameterInput1;
ServerModule.Output.SkillOutput.SkillOutput3.ParameterOutput.ParameterOutput1 := ArrayModule.Output.SkillOutput[3].ParameterOutput[1];
ArrayModule.Input.SkillInput[3].ParameterInput[2] := ServerModule.Input.SkillInput.SkillInput3.ParameterInput.ParameterInput2;
ServerModule.Output.SkillOutput.SkillOutput3.ParameterOutput.ParameterOutput2 := ArrayModule.Output.SkillOutput[3].ParameterOutput[2];
ArrayModule.Input.SkillInput[3].ParameterInput[3] := ServerModule.Input.SkillInput.SkillInput3.ParameterInput.ParameterInput3;
ServerModule.Output.SkillOutput.SkillOutput3.ParameterOutput.ParameterOutput3 := ArrayModule.Output.SkillOutput[3].ParameterOutput[3];
ArrayModule.Input.SkillInput[3].ParameterInput[4] := ServerModule.Input.SkillInput.SkillInput3.ParameterInput.ParameterInput4;
ServerModule.Output.SkillOutput.SkillOutput3.ParameterOutput.ParameterOutput4 := ArrayModule.Output.SkillOutput[3].ParameterOutput[4];
ArrayModule.Input.SkillInput[3].ParameterInput[5] := ServerModule.Input.SkillInput.SkillInput3.ParameterInput.ParameterInput5;
ServerModule.Output.SkillOutput.SkillOutput3.ParameterOutput.ParameterOutput5 := ArrayModule.Output.SkillOutput[3].ParameterOutput[5];
ArrayModule.Input.SkillInput[4].Execute := ServerModule.Input.SkillInput.SkillInput4.Execute;
ServerModule.Output.SkillOutput.SkillOutput4.Dummy := ArrayModule.Output.SkillOutput[4].Dummy;
ServerModule.Output.SkillOutput.SkillOutput4.ID := ArrayModule.Output.SkillOutput[4].ID;
ServerModule.Output.SkillOutput.SkillOutput4.Name := ArrayModule.Output.SkillOutput[4].Name;
ServerModule.Output.SkillOutput.SkillOutput4.Activated := ArrayModule.Output.SkillOutput[4].Activated;
ServerModule.Output.SkillOutput.SkillOutput4.Ready := ArrayModule.Output.SkillOutput[4].Ready;
ServerModule.Output.SkillOutput.SkillOutput4.Busy := ArrayModule.Output.SkillOutput[4].Busy;
ServerModule.Output.SkillOutput.SkillOutput4.Done := ArrayModule.Output.SkillOutput[4].Done;
ServerModule.Output.SkillOutput.SkillOutput4.Error := ArrayModule.Output.SkillOutput[4].Error;
ServerModule.Output.Statevalue.Statevalue0 := ArrayModule.Output.Statevalue[0];
ServerModule.Output.Statevalue.Statevalue1 := ArrayModule.Output.Statevalue[1];
ServerModule.Output.Statevalue.Statevalue2 := ArrayModule.Output.Statevalue[2];
ServerModule.Output.Statevalue.Statevalue3 := ArrayModule.Output.Statevalue[3];
ServerModule.Output.Statevalue.Statevalue4 := ArrayModule.Output.Statevalue[4];
ServerModule.Output.Statevalue.Statevalue5 := ArrayModule.Output.Statevalue[5];
ServerModule.Output.Statevalue.Statevalue6 := ArrayModule.Output.Statevalue[6];
ServerModule.Output.Statevalue.Statevalue7 := ArrayModule.Output.Statevalue[7];
ServerModule.Output.Statevalue.Statevalue8 := ArrayModule.Output.Statevalue[8];
ServerModule.Output.Statevalue.Statevalue9 := ArrayModule.Output.Statevalue[9];
ServerModule.Output.Statevalue.Statevalue10 := ArrayModule.Output.Statevalue[10];
ArrayModule.Input.SkillInput[4].ParameterInput[0] := ServerModule.Input.SkillInput.SkillInput4.ParameterInput.ParameterInput0;
ServerModule.Output.SkillOutput.SkillOutput4.ParameterOutput.ParameterOutput0 := ArrayModule.Output.SkillOutput[4].ParameterOutput[0];
ArrayModule.Input.SkillInput[4].ParameterInput[1] := ServerModule.Input.SkillInput.SkillInput4.ParameterInput.ParameterInput1;
ServerModule.Output.SkillOutput.SkillOutput4.ParameterOutput.ParameterOutput1 := ArrayModule.Output.SkillOutput[4].ParameterOutput[1];
ArrayModule.Input.SkillInput[4].ParameterInput[2] := ServerModule.Input.SkillInput.SkillInput4.ParameterInput.ParameterInput2;
ServerModule.Output.SkillOutput.SkillOutput4.ParameterOutput.ParameterOutput2 := ArrayModule.Output.SkillOutput[4].ParameterOutput[2];
ArrayModule.Input.SkillInput[4].ParameterInput[3] := ServerModule.Input.SkillInput.SkillInput4.ParameterInput.ParameterInput3;
ServerModule.Output.SkillOutput.SkillOutput4.ParameterOutput.ParameterOutput3 := ArrayModule.Output.SkillOutput[4].ParameterOutput[3];
ArrayModule.Input.SkillInput[4].ParameterInput[4] := ServerModule.Input.SkillInput.SkillInput4.ParameterInput.ParameterInput4;
ServerModule.Output.SkillOutput.SkillOutput4.ParameterOutput.ParameterOutput4 := ArrayModule.Output.SkillOutput[4].ParameterOutput[4];
ArrayModule.Input.SkillInput[4].ParameterInput[5] := ServerModule.Input.SkillInput.SkillInput4.ParameterInput.ParameterInput5;
ServerModule.Output.SkillOutput.SkillOutput4.ParameterOutput.ParameterOutput5 := ArrayModule.Output.SkillOutput[4].ParameterOutput[5];
ArrayModule.Input.SkillInput[5].Execute := ServerModule.Input.SkillInput.SkillInput5.Execute;
ServerModule.Output.SkillOutput.SkillOutput5.Dummy := ArrayModule.Output.SkillOutput[5].Dummy;
ServerModule.Output.SkillOutput.SkillOutput5.ID := ArrayModule.Output.SkillOutput[5].ID;
ServerModule.Output.SkillOutput.SkillOutput5.Name := ArrayModule.Output.SkillOutput[5].Name;
ServerModule.Output.SkillOutput.SkillOutput5.Activated := ArrayModule.Output.SkillOutput[5].Activated;
ServerModule.Output.SkillOutput.SkillOutput5.Ready := ArrayModule.Output.SkillOutput[5].Ready;
ServerModule.Output.SkillOutput.SkillOutput5.Busy := ArrayModule.Output.SkillOutput[5].Busy;
ServerModule.Output.SkillOutput.SkillOutput5.Done := ArrayModule.Output.SkillOutput[5].Done;
ServerModule.Output.SkillOutput.SkillOutput5.Error := ArrayModule.Output.SkillOutput[5].Error;
ServerModule.Output.Statevalue.Statevalue0 := ArrayModule.Output.Statevalue[0];
ServerModule.Output.Statevalue.Statevalue1 := ArrayModule.Output.Statevalue[1];
ServerModule.Output.Statevalue.Statevalue2 := ArrayModule.Output.Statevalue[2];
ServerModule.Output.Statevalue.Statevalue3 := ArrayModule.Output.Statevalue[3];
ServerModule.Output.Statevalue.Statevalue4 := ArrayModule.Output.Statevalue[4];
ServerModule.Output.Statevalue.Statevalue5 := ArrayModule.Output.Statevalue[5];
ServerModule.Output.Statevalue.Statevalue6 := ArrayModule.Output.Statevalue[6];
ServerModule.Output.Statevalue.Statevalue7 := ArrayModule.Output.Statevalue[7];
ServerModule.Output.Statevalue.Statevalue8 := ArrayModule.Output.Statevalue[8];
ServerModule.Output.Statevalue.Statevalue9 := ArrayModule.Output.Statevalue[9];
ServerModule.Output.Statevalue.Statevalue10 := ArrayModule.Output.Statevalue[10];
ArrayModule.Input.SkillInput[5].ParameterInput[0] := ServerModule.Input.SkillInput.SkillInput5.ParameterInput.ParameterInput0;
ServerModule.Output.SkillOutput.SkillOutput5.ParameterOutput.ParameterOutput0 := ArrayModule.Output.SkillOutput[5].ParameterOutput[0];
ArrayModule.Input.SkillInput[5].ParameterInput[1] := ServerModule.Input.SkillInput.SkillInput5.ParameterInput.ParameterInput1;
ServerModule.Output.SkillOutput.SkillOutput5.ParameterOutput.ParameterOutput1 := ArrayModule.Output.SkillOutput[5].ParameterOutput[1];
ArrayModule.Input.SkillInput[5].ParameterInput[2] := ServerModule.Input.SkillInput.SkillInput5.ParameterInput.ParameterInput2;
ServerModule.Output.SkillOutput.SkillOutput5.ParameterOutput.ParameterOutput2 := ArrayModule.Output.SkillOutput[5].ParameterOutput[2];
ArrayModule.Input.SkillInput[5].ParameterInput[3] := ServerModule.Input.SkillInput.SkillInput5.ParameterInput.ParameterInput3;
ServerModule.Output.SkillOutput.SkillOutput5.ParameterOutput.ParameterOutput3 := ArrayModule.Output.SkillOutput[5].ParameterOutput[3];
ArrayModule.Input.SkillInput[5].ParameterInput[4] := ServerModule.Input.SkillInput.SkillInput5.ParameterInput.ParameterInput4;
ServerModule.Output.SkillOutput.SkillOutput5.ParameterOutput.ParameterOutput4 := ArrayModule.Output.SkillOutput[5].ParameterOutput[4];
ArrayModule.Input.SkillInput[5].ParameterInput[5] := ServerModule.Input.SkillInput.SkillInput5.ParameterInput.ParameterInput5;
ServerModule.Output.SkillOutput.SkillOutput5.ParameterOutput.ParameterOutput5 := ArrayModule.Output.SkillOutput[5].ParameterOutput[5];
ArrayModule.Input.SkillInput[6].Execute := ServerModule.Input.SkillInput.SkillInput6.Execute;
ServerModule.Output.SkillOutput.SkillOutput6.Dummy := ArrayModule.Output.SkillOutput[6].Dummy;
ServerModule.Output.SkillOutput.SkillOutput6.ID := ArrayModule.Output.SkillOutput[6].ID;
ServerModule.Output.SkillOutput.SkillOutput6.Name := ArrayModule.Output.SkillOutput[6].Name;
ServerModule.Output.SkillOutput.SkillOutput6.Activated := ArrayModule.Output.SkillOutput[6].Activated;
ServerModule.Output.SkillOutput.SkillOutput6.Ready := ArrayModule.Output.SkillOutput[6].Ready;
ServerModule.Output.SkillOutput.SkillOutput6.Busy := ArrayModule.Output.SkillOutput[6].Busy;
ServerModule.Output.SkillOutput.SkillOutput6.Done := ArrayModule.Output.SkillOutput[6].Done;
ServerModule.Output.SkillOutput.SkillOutput6.Error := ArrayModule.Output.SkillOutput[6].Error;
ServerModule.Output.Statevalue.Statevalue0 := ArrayModule.Output.Statevalue[0];
ServerModule.Output.Statevalue.Statevalue1 := ArrayModule.Output.Statevalue[1];
ServerModule.Output.Statevalue.Statevalue2 := ArrayModule.Output.Statevalue[2];
ServerModule.Output.Statevalue.Statevalue3 := ArrayModule.Output.Statevalue[3];
ServerModule.Output.Statevalue.Statevalue4 := ArrayModule.Output.Statevalue[4];
ServerModule.Output.Statevalue.Statevalue5 := ArrayModule.Output.Statevalue[5];
ServerModule.Output.Statevalue.Statevalue6 := ArrayModule.Output.Statevalue[6];
ServerModule.Output.Statevalue.Statevalue7 := ArrayModule.Output.Statevalue[7];
ServerModule.Output.Statevalue.Statevalue8 := ArrayModule.Output.Statevalue[8];
ServerModule.Output.Statevalue.Statevalue9 := ArrayModule.Output.Statevalue[9];
ServerModule.Output.Statevalue.Statevalue10 := ArrayModule.Output.Statevalue[10];
ArrayModule.Input.SkillInput[6].ParameterInput[0] := ServerModule.Input.SkillInput.SkillInput6.ParameterInput.ParameterInput0;
ServerModule.Output.SkillOutput.SkillOutput6.ParameterOutput.ParameterOutput0 := ArrayModule.Output.SkillOutput[6].ParameterOutput[0];
ArrayModule.Input.SkillInput[6].ParameterInput[1] := ServerModule.Input.SkillInput.SkillInput6.ParameterInput.ParameterInput1;
ServerModule.Output.SkillOutput.SkillOutput6.ParameterOutput.ParameterOutput1 := ArrayModule.Output.SkillOutput[6].ParameterOutput[1];
ArrayModule.Input.SkillInput[6].ParameterInput[2] := ServerModule.Input.SkillInput.SkillInput6.ParameterInput.ParameterInput2;
ServerModule.Output.SkillOutput.SkillOutput6.ParameterOutput.ParameterOutput2 := ArrayModule.Output.SkillOutput[6].ParameterOutput[2];
ArrayModule.Input.SkillInput[6].ParameterInput[3] := ServerModule.Input.SkillInput.SkillInput6.ParameterInput.ParameterInput3;
ServerModule.Output.SkillOutput.SkillOutput6.ParameterOutput.ParameterOutput3 := ArrayModule.Output.SkillOutput[6].ParameterOutput[3];
ArrayModule.Input.SkillInput[6].ParameterInput[4] := ServerModule.Input.SkillInput.SkillInput6.ParameterInput.ParameterInput4;
ServerModule.Output.SkillOutput.SkillOutput6.ParameterOutput.ParameterOutput4 := ArrayModule.Output.SkillOutput[6].ParameterOutput[4];
ArrayModule.Input.SkillInput[6].ParameterInput[5] := ServerModule.Input.SkillInput.SkillInput6.ParameterInput.ParameterInput5;
ServerModule.Output.SkillOutput.SkillOutput6.ParameterOutput.ParameterOutput5 := ArrayModule.Output.SkillOutput[6].ParameterOutput[5];
ArrayModule.Input.SkillInput[7].Execute := ServerModule.Input.SkillInput.SkillInput7.Execute;
ServerModule.Output.SkillOutput.SkillOutput7.Dummy := ArrayModule.Output.SkillOutput[7].Dummy;
ServerModule.Output.SkillOutput.SkillOutput7.ID := ArrayModule.Output.SkillOutput[7].ID;
ServerModule.Output.SkillOutput.SkillOutput7.Name := ArrayModule.Output.SkillOutput[7].Name;
ServerModule.Output.SkillOutput.SkillOutput7.Activated := ArrayModule.Output.SkillOutput[7].Activated;
ServerModule.Output.SkillOutput.SkillOutput7.Ready := ArrayModule.Output.SkillOutput[7].Ready;
ServerModule.Output.SkillOutput.SkillOutput7.Busy := ArrayModule.Output.SkillOutput[7].Busy;
ServerModule.Output.SkillOutput.SkillOutput7.Done := ArrayModule.Output.SkillOutput[7].Done;
ServerModule.Output.SkillOutput.SkillOutput7.Error := ArrayModule.Output.SkillOutput[7].Error;
ServerModule.Output.Statevalue.Statevalue0 := ArrayModule.Output.Statevalue[0];
ServerModule.Output.Statevalue.Statevalue1 := ArrayModule.Output.Statevalue[1];
ServerModule.Output.Statevalue.Statevalue2 := ArrayModule.Output.Statevalue[2];
ServerModule.Output.Statevalue.Statevalue3 := ArrayModule.Output.Statevalue[3];
ServerModule.Output.Statevalue.Statevalue4 := ArrayModule.Output.Statevalue[4];
ServerModule.Output.Statevalue.Statevalue5 := ArrayModule.Output.Statevalue[5];
ServerModule.Output.Statevalue.Statevalue6 := ArrayModule.Output.Statevalue[6];
ServerModule.Output.Statevalue.Statevalue7 := ArrayModule.Output.Statevalue[7];
ServerModule.Output.Statevalue.Statevalue8 := ArrayModule.Output.Statevalue[8];
ServerModule.Output.Statevalue.Statevalue9 := ArrayModule.Output.Statevalue[9];
ServerModule.Output.Statevalue.Statevalue10 := ArrayModule.Output.Statevalue[10];
ArrayModule.Input.SkillInput[7].ParameterInput[0] := ServerModule.Input.SkillInput.SkillInput7.ParameterInput.ParameterInput0;
ServerModule.Output.SkillOutput.SkillOutput7.ParameterOutput.ParameterOutput0 := ArrayModule.Output.SkillOutput[7].ParameterOutput[0];
ArrayModule.Input.SkillInput[7].ParameterInput[1] := ServerModule.Input.SkillInput.SkillInput7.ParameterInput.ParameterInput1;
ServerModule.Output.SkillOutput.SkillOutput7.ParameterOutput.ParameterOutput1 := ArrayModule.Output.SkillOutput[7].ParameterOutput[1];
ArrayModule.Input.SkillInput[7].ParameterInput[2] := ServerModule.Input.SkillInput.SkillInput7.ParameterInput.ParameterInput2;
ServerModule.Output.SkillOutput.SkillOutput7.ParameterOutput.ParameterOutput2 := ArrayModule.Output.SkillOutput[7].ParameterOutput[2];
ArrayModule.Input.SkillInput[7].ParameterInput[3] := ServerModule.Input.SkillInput.SkillInput7.ParameterInput.ParameterInput3;
ServerModule.Output.SkillOutput.SkillOutput7.ParameterOutput.ParameterOutput3 := ArrayModule.Output.SkillOutput[7].ParameterOutput[3];
ArrayModule.Input.SkillInput[7].ParameterInput[4] := ServerModule.Input.SkillInput.SkillInput7.ParameterInput.ParameterInput4;
ServerModule.Output.SkillOutput.SkillOutput7.ParameterOutput.ParameterOutput4 := ArrayModule.Output.SkillOutput[7].ParameterOutput[4];
ArrayModule.Input.SkillInput[7].ParameterInput[5] := ServerModule.Input.SkillInput.SkillInput7.ParameterInput.ParameterInput5;
ServerModule.Output.SkillOutput.SkillOutput7.ParameterOutput.ParameterOutput5 := ArrayModule.Output.SkillOutput[7].ParameterOutput[5];
ArrayModule.Input.SkillInput[8].Execute := ServerModule.Input.SkillInput.SkillInput8.Execute;
ServerModule.Output.SkillOutput.SkillOutput8.Dummy := ArrayModule.Output.SkillOutput[8].Dummy;
ServerModule.Output.SkillOutput.SkillOutput8.ID := ArrayModule.Output.SkillOutput[8].ID;
ServerModule.Output.SkillOutput.SkillOutput8.Name := ArrayModule.Output.SkillOutput[8].Name;
ServerModule.Output.SkillOutput.SkillOutput8.Activated := ArrayModule.Output.SkillOutput[8].Activated;
ServerModule.Output.SkillOutput.SkillOutput8.Ready := ArrayModule.Output.SkillOutput[8].Ready;
ServerModule.Output.SkillOutput.SkillOutput8.Busy := ArrayModule.Output.SkillOutput[8].Busy;
ServerModule.Output.SkillOutput.SkillOutput8.Done := ArrayModule.Output.SkillOutput[8].Done;
ServerModule.Output.SkillOutput.SkillOutput8.Error := ArrayModule.Output.SkillOutput[8].Error;
ServerModule.Output.Statevalue.Statevalue0 := ArrayModule.Output.Statevalue[0];
ServerModule.Output.Statevalue.Statevalue1 := ArrayModule.Output.Statevalue[1];
ServerModule.Output.Statevalue.Statevalue2 := ArrayModule.Output.Statevalue[2];
ServerModule.Output.Statevalue.Statevalue3 := ArrayModule.Output.Statevalue[3];
ServerModule.Output.Statevalue.Statevalue4 := ArrayModule.Output.Statevalue[4];
ServerModule.Output.Statevalue.Statevalue5 := ArrayModule.Output.Statevalue[5];
ServerModule.Output.Statevalue.Statevalue6 := ArrayModule.Output.Statevalue[6];
ServerModule.Output.Statevalue.Statevalue7 := ArrayModule.Output.Statevalue[7];
ServerModule.Output.Statevalue.Statevalue8 := ArrayModule.Output.Statevalue[8];
ServerModule.Output.Statevalue.Statevalue9 := ArrayModule.Output.Statevalue[9];
ServerModule.Output.Statevalue.Statevalue10 := ArrayModule.Output.Statevalue[10];
ArrayModule.Input.SkillInput[8].ParameterInput[0] := ServerModule.Input.SkillInput.SkillInput8.ParameterInput.ParameterInput0;
ServerModule.Output.SkillOutput.SkillOutput8.ParameterOutput.ParameterOutput0 := ArrayModule.Output.SkillOutput[8].ParameterOutput[0];
ArrayModule.Input.SkillInput[8].ParameterInput[1] := ServerModule.Input.SkillInput.SkillInput8.ParameterInput.ParameterInput1;
ServerModule.Output.SkillOutput.SkillOutput8.ParameterOutput.ParameterOutput1 := ArrayModule.Output.SkillOutput[8].ParameterOutput[1];
ArrayModule.Input.SkillInput[8].ParameterInput[2] := ServerModule.Input.SkillInput.SkillInput8.ParameterInput.ParameterInput2;
ServerModule.Output.SkillOutput.SkillOutput8.ParameterOutput.ParameterOutput2 := ArrayModule.Output.SkillOutput[8].ParameterOutput[2];
ArrayModule.Input.SkillInput[8].ParameterInput[3] := ServerModule.Input.SkillInput.SkillInput8.ParameterInput.ParameterInput3;
ServerModule.Output.SkillOutput.SkillOutput8.ParameterOutput.ParameterOutput3 := ArrayModule.Output.SkillOutput[8].ParameterOutput[3];
ArrayModule.Input.SkillInput[8].ParameterInput[4] := ServerModule.Input.SkillInput.SkillInput8.ParameterInput.ParameterInput4;
ServerModule.Output.SkillOutput.SkillOutput8.ParameterOutput.ParameterOutput4 := ArrayModule.Output.SkillOutput[8].ParameterOutput[4];
ArrayModule.Input.SkillInput[8].ParameterInput[5] := ServerModule.Input.SkillInput.SkillInput8.ParameterInput.ParameterInput5;
ServerModule.Output.SkillOutput.SkillOutput8.ParameterOutput.ParameterOutput5 := ArrayModule.Output.SkillOutput[8].ParameterOutput[5];
ArrayModule.Input.SkillInput[9].Execute := ServerModule.Input.SkillInput.SkillInput9.Execute;
ServerModule.Output.SkillOutput.SkillOutput9.Dummy := ArrayModule.Output.SkillOutput[9].Dummy;
ServerModule.Output.SkillOutput.SkillOutput9.ID := ArrayModule.Output.SkillOutput[9].ID;
ServerModule.Output.SkillOutput.SkillOutput9.Name := ArrayModule.Output.SkillOutput[9].Name;
ServerModule.Output.SkillOutput.SkillOutput9.Activated := ArrayModule.Output.SkillOutput[9].Activated;
ServerModule.Output.SkillOutput.SkillOutput9.Ready := ArrayModule.Output.SkillOutput[9].Ready;
ServerModule.Output.SkillOutput.SkillOutput9.Busy := ArrayModule.Output.SkillOutput[9].Busy;
ServerModule.Output.SkillOutput.SkillOutput9.Done := ArrayModule.Output.SkillOutput[9].Done;
ServerModule.Output.SkillOutput.SkillOutput9.Error := ArrayModule.Output.SkillOutput[9].Error;
ServerModule.Output.Statevalue.Statevalue0 := ArrayModule.Output.Statevalue[0];
ServerModule.Output.Statevalue.Statevalue1 := ArrayModule.Output.Statevalue[1];
ServerModule.Output.Statevalue.Statevalue2 := ArrayModule.Output.Statevalue[2];
ServerModule.Output.Statevalue.Statevalue3 := ArrayModule.Output.Statevalue[3];
ServerModule.Output.Statevalue.Statevalue4 := ArrayModule.Output.Statevalue[4];
ServerModule.Output.Statevalue.Statevalue5 := ArrayModule.Output.Statevalue[5];
ServerModule.Output.Statevalue.Statevalue6 := ArrayModule.Output.Statevalue[6];
ServerModule.Output.Statevalue.Statevalue7 := ArrayModule.Output.Statevalue[7];
ServerModule.Output.Statevalue.Statevalue8 := ArrayModule.Output.Statevalue[8];
ServerModule.Output.Statevalue.Statevalue9 := ArrayModule.Output.Statevalue[9];
ServerModule.Output.Statevalue.Statevalue10 := ArrayModule.Output.Statevalue[10];
ArrayModule.Input.SkillInput[9].ParameterInput[0] := ServerModule.Input.SkillInput.SkillInput9.ParameterInput.ParameterInput0;
ServerModule.Output.SkillOutput.SkillOutput9.ParameterOutput.ParameterOutput0 := ArrayModule.Output.SkillOutput[9].ParameterOutput[0];
ArrayModule.Input.SkillInput[9].ParameterInput[1] := ServerModule.Input.SkillInput.SkillInput9.ParameterInput.ParameterInput1;
ServerModule.Output.SkillOutput.SkillOutput9.ParameterOutput.ParameterOutput1 := ArrayModule.Output.SkillOutput[9].ParameterOutput[1];
ArrayModule.Input.SkillInput[9].ParameterInput[2] := ServerModule.Input.SkillInput.SkillInput9.ParameterInput.ParameterInput2;
ServerModule.Output.SkillOutput.SkillOutput9.ParameterOutput.ParameterOutput2 := ArrayModule.Output.SkillOutput[9].ParameterOutput[2];
ArrayModule.Input.SkillInput[9].ParameterInput[3] := ServerModule.Input.SkillInput.SkillInput9.ParameterInput.ParameterInput3;
ServerModule.Output.SkillOutput.SkillOutput9.ParameterOutput.ParameterOutput3 := ArrayModule.Output.SkillOutput[9].ParameterOutput[3];
ArrayModule.Input.SkillInput[9].ParameterInput[4] := ServerModule.Input.SkillInput.SkillInput9.ParameterInput.ParameterInput4;
ServerModule.Output.SkillOutput.SkillOutput9.ParameterOutput.ParameterOutput4 := ArrayModule.Output.SkillOutput[9].ParameterOutput[4];
ArrayModule.Input.SkillInput[9].ParameterInput[5] := ServerModule.Input.SkillInput.SkillInput9.ParameterInput.ParameterInput5;
ServerModule.Output.SkillOutput.SkillOutput9.ParameterOutput.ParameterOutput5 := ArrayModule.Output.SkillOutput[9].ParameterOutput[5];
ArrayModule.Input.SkillInput[10].Execute := ServerModule.Input.SkillInput.SkillInput10.Execute;
ServerModule.Output.SkillOutput.SkillOutput10.Dummy := ArrayModule.Output.SkillOutput[10].Dummy;
ServerModule.Output.SkillOutput.SkillOutput10.ID := ArrayModule.Output.SkillOutput[10].ID;
ServerModule.Output.SkillOutput.SkillOutput10.Name := ArrayModule.Output.SkillOutput[10].Name;
ServerModule.Output.SkillOutput.SkillOutput10.Activated := ArrayModule.Output.SkillOutput[10].Activated;
ServerModule.Output.SkillOutput.SkillOutput10.Ready := ArrayModule.Output.SkillOutput[10].Ready;
ServerModule.Output.SkillOutput.SkillOutput10.Busy := ArrayModule.Output.SkillOutput[10].Busy;
ServerModule.Output.SkillOutput.SkillOutput10.Done := ArrayModule.Output.SkillOutput[10].Done;
ServerModule.Output.SkillOutput.SkillOutput10.Error := ArrayModule.Output.SkillOutput[10].Error;
ServerModule.Output.Statevalue.Statevalue0 := ArrayModule.Output.Statevalue[0];
ServerModule.Output.Statevalue.Statevalue1 := ArrayModule.Output.Statevalue[1];
ServerModule.Output.Statevalue.Statevalue2 := ArrayModule.Output.Statevalue[2];
ServerModule.Output.Statevalue.Statevalue3 := ArrayModule.Output.Statevalue[3];
ServerModule.Output.Statevalue.Statevalue4 := ArrayModule.Output.Statevalue[4];
ServerModule.Output.Statevalue.Statevalue5 := ArrayModule.Output.Statevalue[5];
ServerModule.Output.Statevalue.Statevalue6 := ArrayModule.Output.Statevalue[6];
ServerModule.Output.Statevalue.Statevalue7 := ArrayModule.Output.Statevalue[7];
ServerModule.Output.Statevalue.Statevalue8 := ArrayModule.Output.Statevalue[8];
ServerModule.Output.Statevalue.Statevalue9 := ArrayModule.Output.Statevalue[9];
ServerModule.Output.Statevalue.Statevalue10 := ArrayModule.Output.Statevalue[10];
ArrayModule.Input.SkillInput[10].ParameterInput[0] := ServerModule.Input.SkillInput.SkillInput10.ParameterInput.ParameterInput0;
ServerModule.Output.SkillOutput.SkillOutput10.ParameterOutput.ParameterOutput0 := ArrayModule.Output.SkillOutput[10].ParameterOutput[0];
ArrayModule.Input.SkillInput[10].ParameterInput[1] := ServerModule.Input.SkillInput.SkillInput10.ParameterInput.ParameterInput1;
ServerModule.Output.SkillOutput.SkillOutput10.ParameterOutput.ParameterOutput1 := ArrayModule.Output.SkillOutput[10].ParameterOutput[1];
ArrayModule.Input.SkillInput[10].ParameterInput[2] := ServerModule.Input.SkillInput.SkillInput10.ParameterInput.ParameterInput2;
ServerModule.Output.SkillOutput.SkillOutput10.ParameterOutput.ParameterOutput2 := ArrayModule.Output.SkillOutput[10].ParameterOutput[2];
ArrayModule.Input.SkillInput[10].ParameterInput[3] := ServerModule.Input.SkillInput.SkillInput10.ParameterInput.ParameterInput3;
ServerModule.Output.SkillOutput.SkillOutput10.ParameterOutput.ParameterOutput3 := ArrayModule.Output.SkillOutput[10].ParameterOutput[3];
ArrayModule.Input.SkillInput[10].ParameterInput[4] := ServerModule.Input.SkillInput.SkillInput10.ParameterInput.ParameterInput4;
ServerModule.Output.SkillOutput.SkillOutput10.ParameterOutput.ParameterOutput4 := ArrayModule.Output.SkillOutput[10].ParameterOutput[4];
ArrayModule.Input.SkillInput[10].ParameterInput[5] := ServerModule.Input.SkillInput.SkillInput10.ParameterInput.ParameterInput5;
ServerModule.Output.SkillOutput.SkillOutput10.ParameterOutput.ParameterOutput5 := ArrayModule.Output.SkillOutput[10].ParameterOutput[5];
ArrayModule.Input.SkillInput[11].Execute := ServerModule.Input.SkillInput.SkillInput11.Execute;
ServerModule.Output.SkillOutput.SkillOutput11.Dummy := ArrayModule.Output.SkillOutput[11].Dummy;
ServerModule.Output.SkillOutput.SkillOutput11.ID := ArrayModule.Output.SkillOutput[11].ID;
ServerModule.Output.SkillOutput.SkillOutput11.Name := ArrayModule.Output.SkillOutput[11].Name;
ServerModule.Output.SkillOutput.SkillOutput11.Activated := ArrayModule.Output.SkillOutput[11].Activated;
ServerModule.Output.SkillOutput.SkillOutput11.Ready := ArrayModule.Output.SkillOutput[11].Ready;
ServerModule.Output.SkillOutput.SkillOutput11.Busy := ArrayModule.Output.SkillOutput[11].Busy;
ServerModule.Output.SkillOutput.SkillOutput11.Done := ArrayModule.Output.SkillOutput[11].Done;
ServerModule.Output.SkillOutput.SkillOutput11.Error := ArrayModule.Output.SkillOutput[11].Error;
ServerModule.Output.Statevalue.Statevalue0 := ArrayModule.Output.Statevalue[0];
ServerModule.Output.Statevalue.Statevalue1 := ArrayModule.Output.Statevalue[1];
ServerModule.Output.Statevalue.Statevalue2 := ArrayModule.Output.Statevalue[2];
ServerModule.Output.Statevalue.Statevalue3 := ArrayModule.Output.Statevalue[3];
ServerModule.Output.Statevalue.Statevalue4 := ArrayModule.Output.Statevalue[4];
ServerModule.Output.Statevalue.Statevalue5 := ArrayModule.Output.Statevalue[5];
ServerModule.Output.Statevalue.Statevalue6 := ArrayModule.Output.Statevalue[6];
ServerModule.Output.Statevalue.Statevalue7 := ArrayModule.Output.Statevalue[7];
ServerModule.Output.Statevalue.Statevalue8 := ArrayModule.Output.Statevalue[8];
ServerModule.Output.Statevalue.Statevalue9 := ArrayModule.Output.Statevalue[9];
ServerModule.Output.Statevalue.Statevalue10 := ArrayModule.Output.Statevalue[10];
ArrayModule.Input.SkillInput[11].ParameterInput[0] := ServerModule.Input.SkillInput.SkillInput11.ParameterInput.ParameterInput0;
ServerModule.Output.SkillOutput.SkillOutput11.ParameterOutput.ParameterOutput0 := ArrayModule.Output.SkillOutput[11].ParameterOutput[0];
ArrayModule.Input.SkillInput[11].ParameterInput[1] := ServerModule.Input.SkillInput.SkillInput11.ParameterInput.ParameterInput1;
ServerModule.Output.SkillOutput.SkillOutput11.ParameterOutput.ParameterOutput1 := ArrayModule.Output.SkillOutput[11].ParameterOutput[1];
ArrayModule.Input.SkillInput[11].ParameterInput[2] := ServerModule.Input.SkillInput.SkillInput11.ParameterInput.ParameterInput2;
ServerModule.Output.SkillOutput.SkillOutput11.ParameterOutput.ParameterOutput2 := ArrayModule.Output.SkillOutput[11].ParameterOutput[2];
ArrayModule.Input.SkillInput[11].ParameterInput[3] := ServerModule.Input.SkillInput.SkillInput11.ParameterInput.ParameterInput3;
ServerModule.Output.SkillOutput.SkillOutput11.ParameterOutput.ParameterOutput3 := ArrayModule.Output.SkillOutput[11].ParameterOutput[3];
ArrayModule.Input.SkillInput[11].ParameterInput[4] := ServerModule.Input.SkillInput.SkillInput11.ParameterInput.ParameterInput4;
ServerModule.Output.SkillOutput.SkillOutput11.ParameterOutput.ParameterOutput4 := ArrayModule.Output.SkillOutput[11].ParameterOutput[4];
ArrayModule.Input.SkillInput[11].ParameterInput[5] := ServerModule.Input.SkillInput.SkillInput11.ParameterInput.ParameterInput5;
ServerModule.Output.SkillOutput.SkillOutput11.ParameterOutput.ParameterOutput5 := ArrayModule.Output.SkillOutput[11].ParameterOutput[5];
ArrayModule.Input.SkillInput[12].Execute := ServerModule.Input.SkillInput.SkillInput12.Execute;
ServerModule.Output.SkillOutput.SkillOutput12.Dummy := ArrayModule.Output.SkillOutput[12].Dummy;
ServerModule.Output.SkillOutput.SkillOutput12.ID := ArrayModule.Output.SkillOutput[12].ID;
ServerModule.Output.SkillOutput.SkillOutput12.Name := ArrayModule.Output.SkillOutput[12].Name;
ServerModule.Output.SkillOutput.SkillOutput12.Activated := ArrayModule.Output.SkillOutput[12].Activated;
ServerModule.Output.SkillOutput.SkillOutput12.Ready := ArrayModule.Output.SkillOutput[12].Ready;
ServerModule.Output.SkillOutput.SkillOutput12.Busy := ArrayModule.Output.SkillOutput[12].Busy;
ServerModule.Output.SkillOutput.SkillOutput12.Done := ArrayModule.Output.SkillOutput[12].Done;
ServerModule.Output.SkillOutput.SkillOutput12.Error := ArrayModule.Output.SkillOutput[12].Error;
ServerModule.Output.Statevalue.Statevalue0 := ArrayModule.Output.Statevalue[0];
ServerModule.Output.Statevalue.Statevalue1 := ArrayModule.Output.Statevalue[1];
ServerModule.Output.Statevalue.Statevalue2 := ArrayModule.Output.Statevalue[2];
ServerModule.Output.Statevalue.Statevalue3 := ArrayModule.Output.Statevalue[3];
ServerModule.Output.Statevalue.Statevalue4 := ArrayModule.Output.Statevalue[4];
ServerModule.Output.Statevalue.Statevalue5 := ArrayModule.Output.Statevalue[5];
ServerModule.Output.Statevalue.Statevalue6 := ArrayModule.Output.Statevalue[6];
ServerModule.Output.Statevalue.Statevalue7 := ArrayModule.Output.Statevalue[7];
ServerModule.Output.Statevalue.Statevalue8 := ArrayModule.Output.Statevalue[8];
ServerModule.Output.Statevalue.Statevalue9 := ArrayModule.Output.Statevalue[9];
ServerModule.Output.Statevalue.Statevalue10 := ArrayModule.Output.Statevalue[10];
ArrayModule.Input.SkillInput[12].ParameterInput[0] := ServerModule.Input.SkillInput.SkillInput12.ParameterInput.ParameterInput0;
ServerModule.Output.SkillOutput.SkillOutput12.ParameterOutput.ParameterOutput0 := ArrayModule.Output.SkillOutput[12].ParameterOutput[0];
ArrayModule.Input.SkillInput[12].ParameterInput[1] := ServerModule.Input.SkillInput.SkillInput12.ParameterInput.ParameterInput1;
ServerModule.Output.SkillOutput.SkillOutput12.ParameterOutput.ParameterOutput1 := ArrayModule.Output.SkillOutput[12].ParameterOutput[1];
ArrayModule.Input.SkillInput[12].ParameterInput[2] := ServerModule.Input.SkillInput.SkillInput12.ParameterInput.ParameterInput2;
ServerModule.Output.SkillOutput.SkillOutput12.ParameterOutput.ParameterOutput2 := ArrayModule.Output.SkillOutput[12].ParameterOutput[2];
ArrayModule.Input.SkillInput[12].ParameterInput[3] := ServerModule.Input.SkillInput.SkillInput12.ParameterInput.ParameterInput3;
ServerModule.Output.SkillOutput.SkillOutput12.ParameterOutput.ParameterOutput3 := ArrayModule.Output.SkillOutput[12].ParameterOutput[3];
ArrayModule.Input.SkillInput[12].ParameterInput[4] := ServerModule.Input.SkillInput.SkillInput12.ParameterInput.ParameterInput4;
ServerModule.Output.SkillOutput.SkillOutput12.ParameterOutput.ParameterOutput4 := ArrayModule.Output.SkillOutput[12].ParameterOutput[4];
ArrayModule.Input.SkillInput[12].ParameterInput[5] := ServerModule.Input.SkillInput.SkillInput12.ParameterInput.ParameterInput5;
ServerModule.Output.SkillOutput.SkillOutput12.ParameterOutput.ParameterOutput5 := ArrayModule.Output.SkillOutput[12].ParameterOutput[5];
ArrayModule.Input.SkillInput[13].Execute := ServerModule.Input.SkillInput.SkillInput13.Execute;
ServerModule.Output.SkillOutput.SkillOutput13.Dummy := ArrayModule.Output.SkillOutput[13].Dummy;
ServerModule.Output.SkillOutput.SkillOutput13.ID := ArrayModule.Output.SkillOutput[13].ID;
ServerModule.Output.SkillOutput.SkillOutput13.Name := ArrayModule.Output.SkillOutput[13].Name;
ServerModule.Output.SkillOutput.SkillOutput13.Activated := ArrayModule.Output.SkillOutput[13].Activated;
ServerModule.Output.SkillOutput.SkillOutput13.Ready := ArrayModule.Output.SkillOutput[13].Ready;
ServerModule.Output.SkillOutput.SkillOutput13.Busy := ArrayModule.Output.SkillOutput[13].Busy;
ServerModule.Output.SkillOutput.SkillOutput13.Done := ArrayModule.Output.SkillOutput[13].Done;
ServerModule.Output.SkillOutput.SkillOutput13.Error := ArrayModule.Output.SkillOutput[13].Error;
ServerModule.Output.Statevalue.Statevalue0 := ArrayModule.Output.Statevalue[0];
ServerModule.Output.Statevalue.Statevalue1 := ArrayModule.Output.Statevalue[1];
ServerModule.Output.Statevalue.Statevalue2 := ArrayModule.Output.Statevalue[2];
ServerModule.Output.Statevalue.Statevalue3 := ArrayModule.Output.Statevalue[3];
ServerModule.Output.Statevalue.Statevalue4 := ArrayModule.Output.Statevalue[4];
ServerModule.Output.Statevalue.Statevalue5 := ArrayModule.Output.Statevalue[5];
ServerModule.Output.Statevalue.Statevalue6 := ArrayModule.Output.Statevalue[6];
ServerModule.Output.Statevalue.Statevalue7 := ArrayModule.Output.Statevalue[7];
ServerModule.Output.Statevalue.Statevalue8 := ArrayModule.Output.Statevalue[8];
ServerModule.Output.Statevalue.Statevalue9 := ArrayModule.Output.Statevalue[9];
ServerModule.Output.Statevalue.Statevalue10 := ArrayModule.Output.Statevalue[10];
ArrayModule.Input.SkillInput[13].ParameterInput[0] := ServerModule.Input.SkillInput.SkillInput13.ParameterInput.ParameterInput0;
ServerModule.Output.SkillOutput.SkillOutput13.ParameterOutput.ParameterOutput0 := ArrayModule.Output.SkillOutput[13].ParameterOutput[0];
ArrayModule.Input.SkillInput[13].ParameterInput[1] := ServerModule.Input.SkillInput.SkillInput13.ParameterInput.ParameterInput1;
ServerModule.Output.SkillOutput.SkillOutput13.ParameterOutput.ParameterOutput1 := ArrayModule.Output.SkillOutput[13].ParameterOutput[1];
ArrayModule.Input.SkillInput[13].ParameterInput[2] := ServerModule.Input.SkillInput.SkillInput13.ParameterInput.ParameterInput2;
ServerModule.Output.SkillOutput.SkillOutput13.ParameterOutput.ParameterOutput2 := ArrayModule.Output.SkillOutput[13].ParameterOutput[2];
ArrayModule.Input.SkillInput[13].ParameterInput[3] := ServerModule.Input.SkillInput.SkillInput13.ParameterInput.ParameterInput3;
ServerModule.Output.SkillOutput.SkillOutput13.ParameterOutput.ParameterOutput3 := ArrayModule.Output.SkillOutput[13].ParameterOutput[3];
ArrayModule.Input.SkillInput[13].ParameterInput[4] := ServerModule.Input.SkillInput.SkillInput13.ParameterInput.ParameterInput4;
ServerModule.Output.SkillOutput.SkillOutput13.ParameterOutput.ParameterOutput4 := ArrayModule.Output.SkillOutput[13].ParameterOutput[4];
ArrayModule.Input.SkillInput[13].ParameterInput[5] := ServerModule.Input.SkillInput.SkillInput13.ParameterInput.ParameterInput5;
ServerModule.Output.SkillOutput.SkillOutput13.ParameterOutput.ParameterOutput5 := ArrayModule.Output.SkillOutput[13].ParameterOutput[5];
ArrayModule.Input.SkillInput[14].Execute := ServerModule.Input.SkillInput.SkillInput14.Execute;
ServerModule.Output.SkillOutput.SkillOutput14.Dummy := ArrayModule.Output.SkillOutput[14].Dummy;
ServerModule.Output.SkillOutput.SkillOutput14.ID := ArrayModule.Output.SkillOutput[14].ID;
ServerModule.Output.SkillOutput.SkillOutput14.Name := ArrayModule.Output.SkillOutput[14].Name;
ServerModule.Output.SkillOutput.SkillOutput14.Activated := ArrayModule.Output.SkillOutput[14].Activated;
ServerModule.Output.SkillOutput.SkillOutput14.Ready := ArrayModule.Output.SkillOutput[14].Ready;
ServerModule.Output.SkillOutput.SkillOutput14.Busy := ArrayModule.Output.SkillOutput[14].Busy;
ServerModule.Output.SkillOutput.SkillOutput14.Done := ArrayModule.Output.SkillOutput[14].Done;
ServerModule.Output.SkillOutput.SkillOutput14.Error := ArrayModule.Output.SkillOutput[14].Error;
ServerModule.Output.Statevalue.Statevalue0 := ArrayModule.Output.Statevalue[0];
ServerModule.Output.Statevalue.Statevalue1 := ArrayModule.Output.Statevalue[1];
ServerModule.Output.Statevalue.Statevalue2 := ArrayModule.Output.Statevalue[2];
ServerModule.Output.Statevalue.Statevalue3 := ArrayModule.Output.Statevalue[3];
ServerModule.Output.Statevalue.Statevalue4 := ArrayModule.Output.Statevalue[4];
ServerModule.Output.Statevalue.Statevalue5 := ArrayModule.Output.Statevalue[5];
ServerModule.Output.Statevalue.Statevalue6 := ArrayModule.Output.Statevalue[6];
ServerModule.Output.Statevalue.Statevalue7 := ArrayModule.Output.Statevalue[7];
ServerModule.Output.Statevalue.Statevalue8 := ArrayModule.Output.Statevalue[8];
ServerModule.Output.Statevalue.Statevalue9 := ArrayModule.Output.Statevalue[9];
ServerModule.Output.Statevalue.Statevalue10 := ArrayModule.Output.Statevalue[10];
ArrayModule.Input.SkillInput[14].ParameterInput[0] := ServerModule.Input.SkillInput.SkillInput14.ParameterInput.ParameterInput0;
ServerModule.Output.SkillOutput.SkillOutput14.ParameterOutput.ParameterOutput0 := ArrayModule.Output.SkillOutput[14].ParameterOutput[0];
ArrayModule.Input.SkillInput[14].ParameterInput[1] := ServerModule.Input.SkillInput.SkillInput14.ParameterInput.ParameterInput1;
ServerModule.Output.SkillOutput.SkillOutput14.ParameterOutput.ParameterOutput1 := ArrayModule.Output.SkillOutput[14].ParameterOutput[1];
ArrayModule.Input.SkillInput[14].ParameterInput[2] := ServerModule.Input.SkillInput.SkillInput14.ParameterInput.ParameterInput2;
ServerModule.Output.SkillOutput.SkillOutput14.ParameterOutput.ParameterOutput2 := ArrayModule.Output.SkillOutput[14].ParameterOutput[2];
ArrayModule.Input.SkillInput[14].ParameterInput[3] := ServerModule.Input.SkillInput.SkillInput14.ParameterInput.ParameterInput3;
ServerModule.Output.SkillOutput.SkillOutput14.ParameterOutput.ParameterOutput3 := ArrayModule.Output.SkillOutput[14].ParameterOutput[3];
ArrayModule.Input.SkillInput[14].ParameterInput[4] := ServerModule.Input.SkillInput.SkillInput14.ParameterInput.ParameterInput4;
ServerModule.Output.SkillOutput.SkillOutput14.ParameterOutput.ParameterOutput4 := ArrayModule.Output.SkillOutput[14].ParameterOutput[4];
ArrayModule.Input.SkillInput[14].ParameterInput[5] := ServerModule.Input.SkillInput.SkillInput14.ParameterInput.ParameterInput5;
ServerModule.Output.SkillOutput.SkillOutput14.ParameterOutput.ParameterOutput5 := ArrayModule.Output.SkillOutput[14].ParameterOutput[5];
ArrayModule.Input.SkillInput[15].Execute := ServerModule.Input.SkillInput.SkillInput15.Execute;
ServerModule.Output.SkillOutput.SkillOutput15.Dummy := ArrayModule.Output.SkillOutput[15].Dummy;
ServerModule.Output.SkillOutput.SkillOutput15.ID := ArrayModule.Output.SkillOutput[15].ID;
ServerModule.Output.SkillOutput.SkillOutput15.Name := ArrayModule.Output.SkillOutput[15].Name;
ServerModule.Output.SkillOutput.SkillOutput15.Activated := ArrayModule.Output.SkillOutput[15].Activated;
ServerModule.Output.SkillOutput.SkillOutput15.Ready := ArrayModule.Output.SkillOutput[15].Ready;
ServerModule.Output.SkillOutput.SkillOutput15.Busy := ArrayModule.Output.SkillOutput[15].Busy;
ServerModule.Output.SkillOutput.SkillOutput15.Done := ArrayModule.Output.SkillOutput[15].Done;
ServerModule.Output.SkillOutput.SkillOutput15.Error := ArrayModule.Output.SkillOutput[15].Error;
ServerModule.Output.Statevalue.Statevalue0 := ArrayModule.Output.Statevalue[0];
ServerModule.Output.Statevalue.Statevalue1 := ArrayModule.Output.Statevalue[1];
ServerModule.Output.Statevalue.Statevalue2 := ArrayModule.Output.Statevalue[2];
ServerModule.Output.Statevalue.Statevalue3 := ArrayModule.Output.Statevalue[3];
ServerModule.Output.Statevalue.Statevalue4 := ArrayModule.Output.Statevalue[4];
ServerModule.Output.Statevalue.Statevalue5 := ArrayModule.Output.Statevalue[5];
ServerModule.Output.Statevalue.Statevalue6 := ArrayModule.Output.Statevalue[6];
ServerModule.Output.Statevalue.Statevalue7 := ArrayModule.Output.Statevalue[7];
ServerModule.Output.Statevalue.Statevalue8 := ArrayModule.Output.Statevalue[8];
ServerModule.Output.Statevalue.Statevalue9 := ArrayModule.Output.Statevalue[9];
ServerModule.Output.Statevalue.Statevalue10 := ArrayModule.Output.Statevalue[10];
ArrayModule.Input.SkillInput[15].ParameterInput[0] := ServerModule.Input.SkillInput.SkillInput15.ParameterInput.ParameterInput0;
ServerModule.Output.SkillOutput.SkillOutput15.ParameterOutput.ParameterOutput0 := ArrayModule.Output.SkillOutput[15].ParameterOutput[0];
ArrayModule.Input.SkillInput[15].ParameterInput[1] := ServerModule.Input.SkillInput.SkillInput15.ParameterInput.ParameterInput1;
ServerModule.Output.SkillOutput.SkillOutput15.ParameterOutput.ParameterOutput1 := ArrayModule.Output.SkillOutput[15].ParameterOutput[1];
ArrayModule.Input.SkillInput[15].ParameterInput[2] := ServerModule.Input.SkillInput.SkillInput15.ParameterInput.ParameterInput2;
ServerModule.Output.SkillOutput.SkillOutput15.ParameterOutput.ParameterOutput2 := ArrayModule.Output.SkillOutput[15].ParameterOutput[2];
ArrayModule.Input.SkillInput[15].ParameterInput[3] := ServerModule.Input.SkillInput.SkillInput15.ParameterInput.ParameterInput3;
ServerModule.Output.SkillOutput.SkillOutput15.ParameterOutput.ParameterOutput3 := ArrayModule.Output.SkillOutput[15].ParameterOutput[3];
ArrayModule.Input.SkillInput[15].ParameterInput[4] := ServerModule.Input.SkillInput.SkillInput15.ParameterInput.ParameterInput4;
ServerModule.Output.SkillOutput.SkillOutput15.ParameterOutput.ParameterOutput4 := ArrayModule.Output.SkillOutput[15].ParameterOutput[4];
ArrayModule.Input.SkillInput[15].ParameterInput[5] := ServerModule.Input.SkillInput.SkillInput15.ParameterInput.ParameterInput5;
ServerModule.Output.SkillOutput.SkillOutput15.ParameterOutput.ParameterOutput5 := ArrayModule.Output.SkillOutput[15].ParameterOutput[5];

END_IF

END_FUNCTION_BLOCK

// ---- POUs/FB_FAKE_MODULE.TcPOU
FUNCTION_BLOCK FB_FAKE_MODULE
VAR_INPUT
	Execute : BOOL;
	SKILLID	: ARRAY [0..SkillCnt] OF INT;
	INPUT	: DUT_MODULE_INTERFACE_INPUT;
	SkillTime	: TIME := T#5S;
	ForceError	: BOOL;
	ID			: INT := 42424;
END_VAR
VAR_OUTPUT
	OUTPUT 	: DUT_MODULE_INTERFACE_OUTPUT;
END_VAR

VAR
	LampTime	: TIME;
	i 		: INT := 0;
	state 	: INT := -10;
	activeNr	: INT;
	TIMER	: TON;
	LampTimer	: TON;
	
	fbi_Timer: TOF;
END_VAR

IF Execute THEN
	CASE state OF
		
	
	-10: 
		OUTPUT.Dummy := FALSE;
		OUTPUT.Name	 := 'BeispielModul';
		OUTPUT.ID	 := ID;
		
		FOR i := 0 TO SkillCnt DO
		
			IF SKILLID[i] > 0 THEN
				OUTPUT.SkillOutput[i].ID := SKILLID[i];
				OUTPUT.SkillOutput[i].Dummy := FALSE;
			END_IF
		
		END_FOR
		state := 0;
		
		
	0: 	// ALLE SKILLS READY
		FOR i := 0 TO SkillCnt DO
			IF SKILLID[i] > 0 THEN 
			OUTPUT.SkillOutput[i].Ready := TRUE;
			OUTPUT.SkillOutput[i].Busy 	:= FALSE;
			OUTPUT.SkillOutput[i].Done 	:= FALSE;
			OUTPUT.SkillOutput[i].Name  := CONCAT ('Beispielskill', INT_TO_STRING(SKILLID[i]));
				IF INPUT.SkillInput[i].Execute THEN
					IF NOT (Input.SkillInput[i].ParameterInput[0].Value = 0) THEN
					LampTime := REAL_TO_TIME(1/Input.SkillInput[i].ParameterInput[0].Value * 1000);
					ELSE
					LampTime := T#1s;
					END_IF
					activeNr := i;
					state := 10;
				END_IF
			END_IF
		END_FOR
		
	10: // KEIN SKILL READY, skill activeNR busy
		FOR i := 0 TO SkillCnt DO
			OUTPUT.SkillOutput[i].Ready := FALSE;		
		END_FOR
			
		OUTPUT.SkillOutput[activeNr].Busy 	:= TRUE;
		OUTPUT.SkillOutput[activeNr].Done 	:= FALSE;
		TIMER(IN := FALSE, PT := SkillTime);
		LampTimer(IN := FALSE, PT := LampTime);
		
		state := 20;
		
	20:	// SKILL AUSFÜHREN
		TIMER(IN := TRUE);
		
		Lamp2 := TRUE;
		LampTimer(IN := TRUE);
		IF LampTimer.Q THEN
			
			LampTimer(IN := FALSE);
			Lamp1 := NOT (Lamp1);
		END_IF
		
		
		
		IF TIMER.Q THEN
			IF NOT ForceError THEN
				OUTPUT.SkillOutput[activeNr].Done 	:= TRUE;
				OUTPUT.SkillOutput[activeNr].Busy	:= FALSE;
			ELSE
				OUTPUT.SkillOutput[activeNr].Error	:= TRUE;
				OUTPUT.SkillOutput[activeNr].Busy	:= FALSE;
			END_IF
			state := 30;
			Lamp2 := FALSE;
			Lamp1 := FALSE;
		END_IF
		
	30: // warten bis execute zurückgezogen
		IF NOT INPUT.SkillInput[activeNr].Execute THEN
			OUTPUT.SkillOutput[activeNr].Done 	:= FALSE;
			OUTPUT.SkillOutput[activeNr].Error	:= FALSE;
			state := 0;
		END_IF
		
	
	
	
	
	END_CASE
ELSE
	state := -10;
END_IF

fbi_Timer();
IF GVL.init_sensor_x THEN
	Output.PositionSensor := TRUE;
	
	fbi_Timer(IN := TRUE,PT := T#400MS);
	fbi_Timer(IN := FALSE,PT := T#400MS);	
ELSE
	Output.PositionSensor := fbi_Timer.Q;
END_IF

Output.ConnectionTestOutput := INPUT.ConnectionTestInput;
OUTPUT.PositionOutput	:= INPUT.PositionInput;

END_FUNCTION_BLOCK

// ---- POUs/industrialPhysics/MAIN_simu.TcPOU

PROGRAM MAIN_simu
VAR
    simIO : MNG_Simulation;
END_VAR

// Update IOs with simulation
simIO(bEnable := TRUE);

// Application code follows here:

END_PROGRAM

// ---- POUs/industrialPhysics/MNG_SIMULATION.TcPOU
FUNCTION_BLOCK MNG_Simulation
VAR_INPUT
    bEnable    : BOOL                          := FALSE;
    outputs    : MNG_APPLICATION_OUTPUTS_32BIT         ;
END_VAR
VAR_OUTPUT
    inputs     : MNG_APPLICATION_INPUTS_32BIT          ;
END_VAR
VAR
    ioUpdater  : MNG_UpdateIOs                 := (sRemoteHost := '192.168.42.31', nRemotePort := 6000);
    fbCloseAll : FB_SocketCloseAll;
    bCloseAll  : BOOL := TRUE;
END_VAR

(* @END_DECLARATION := '0'                                                    *)
IF bCloseAll THEN (*On PLC reset or program download close all old (opened) connections *)
    bCloseAll := FALSE;
    fbCloseAll( bExecute:= TRUE );
ELSE
    fbCloseAll( bExecute:= FALSE );
END_IF

IF NOT fbCloseAll.bBusy THEN

    (* ------------------------------------- trigger data exchange ----------------------------------------------------------------------------*)
   ioUpdater(Outputs := outputs, Inputs => inputs, bEnable := bEnable);

END_IF

outputs.DosierModul_00_ACT_POS02 := (Simulation.XPosition3 -2000)/1000;

outputs.Keksmodul_00_ACT_POS02 := (Simulation.XPosition0 -2000)/1000;

outputs.Toppingmodul_Beckhoff_00_ACT_POS02 := (Simulation.XPosition1 -2000)/1000;

outputs.Toppingmodul_Bosch_00_ACT_POS02 := (Simulation.XPosition2 -2000)/1000;

GVL.init_sensor_x := inputs.init_sensor_module_x_00_IR;

outputs.MotorX_00_par1 := GVL.lamp1;
outputs.MotorX_00_par2 := GVL.lamp2;

outputs.status_00_on102 := MI5.Simulation.Cookie.Ready;
outputs.status_00_on202 := MI5.Simulation.Cookie.Busy;
outputs.status_00_on302 := MI5.Simulation.Cookie.Error;

outputs.status_00_on103 := MI5.Simulation.Topping_Bosch.Ready;
outputs.status_00_on203 := MI5.Simulation.Topping_Bosch.Busy;
outputs.status_00_on303 := MI5.Simulation.Topping_Bosch.Error;

outputs.status_00_on104 := MI5.Simulation.Topping_Beckhoff.Ready;
outputs.status_00_on204 := MI5.Simulation.Topping_Beckhoff.Busy;
outputs.status_00_on304 := MI5.Simulation.Topping_Beckhoff.Error;

outputs.status_00_on105 := MI5.Simulation.Cocktail.Ready;
outputs.status_00_on205 := MI5.Simulation.Cocktail.Busy;
outputs.status_00_on305 := MI5.Simulation.Cocktail.Error;

END_FUNCTION_BLOCK

// ---- POUs/industrialPhysics/MNG_UPDATEIOS.TcPOU
FUNCTION_BLOCK MNG_UpdateIOs
(* This function block implements simple TCP/IP client protocol.              *)
(* The max. size of binary tx/rx data has to be <= PLCPRJ_BUFFER_SIZE         *)
VAR_IN_OUT
    Outputs : MNG_APPLICATION_OUTPUTS_32BIT;    (* Tx user data *)

END_VAR

VAR_INPUT
    bDbg        : BOOL                         := FALSE               ; (* TRUE => Enable debug output, FALSE => Disable debug output *)
    sRemoteHost : STRING(15)                   := '127.0.0.1'         ; (* IP address of remote server *)	
    nRemotePort : UDINT                        := 5000                ; (* Remote server port *)
    bEnable     : BOOL                         := FALSE               ; (* TRUE => Enable/connect, FALSE => Disable/disconnect *)
    tReconnect  : TIME                         := T#5s                ;
END_VAR

VAR_OUTPUT
    errors      : FB_LogFifo                                          ; (* Error message fifo *)
    eState      : E_SocketConnectionState      := eSOCKET_DISCONNECTED; (* TCP/IP connection state *)
    Inputs      : MNG_APPLICATION_INPUTS_32BIT                        ; (* Rx user data *)
END_VAR

VAR
    counter          : DWORD                        := 0                   ;
    fbConnect        : FB_ClientServerConnection    := (tReconnect := T#5s); (* Create/release TCP/IP connection *)
    fbSend           : FB_SocketSend                                       ; (* Send TCP/IP data *)
    fbReceive        : FB_SocketReceive                                    ; (* Receive TCP/IP data *)
    state            : BYTE                                                ; (* Global state *)
    tx_state         : BYTE                                                ; (* Tx state *)
    rx_state         : BYTE                                                ; (* Rx state *)

    toServer         : MNG_RawDatagram                                     ;
    fromServer       : MNG_RawDatagram                                     ;
    cbReceived       : UDINT                                               ; (* Count of received data bytes *)
    cbRx             : UDINT                                               ; (* Rx frame byte size *)

    bDisconnect      : BOOL                                                ; (* Disconnect flag, if set the socket will be closed *)
    pollTimer        : TON                                                 ; (* Rx data poll timer *)
    bAbort           : BOOL                                                ; (* Flag to abort frame parsing loop *)
    sID              : STRING(20)                   := ''                  ;
    clock            : FB_LocalSystemTime           := ( bEnable := TRUE ) ; (* OS clock *)
    _byteCount       : DWORD                                               ;
    _i               : DWORD                                               ;
    _ptr             : POINTER TO BYTE                                     ;
    _internalInputs  : MNG_APPLICATION_INPUTS_32BIT                       ;
    DWordBuffer      : DWORD                                               ; (* convert DWORD data *)
    DIntBuffer       : DINT                                                ; (* convert DINT data *)
END_VAR


(* refresh clock time                                                         *)
clock();

(* state chart                                                                *)
CASE state OF
    0:(* Init state *)
        (*rx.A_Reset(bDbg := bDbg)  ; (* Reset RX fifo (optional) *)
        tx.A_Reset    (bDbg := bDbg); (* Reset TX fifo (optional) *)*)
        errors.Clear(); (* Reset error fifo (optional) *)

        pollTimer( IN := FALSE, PT := PLCPRJ_RECEIVER_POLLING_CYCLE_TIME );
        bDisconnect := FALSE;(* Reset disconnect flag *)
        cbReceived  := 0;(* Reset number of received data bytes *)
        tx_state    := 0;(* Reset tx state machine *)
        rx_state    := 0;(* Reset rx state machine *)
        state       := 1;(* Go to the next step *)

    1:(* Create TCP/IP connection *)
        fbConnect(sSrvNetID := '',
                  nMode := CONNECT_MODE_ENABLEDBG,(* Enable debug output *)
                  sRemoteHost := sRemoteHost,
                  nRemotePort := nRemotePort,
                  tReconnect  := tReconnect,
                  bEnable     := bEnable,
                  eState      => eState);
        IF NOT fbConnect.bBusy THEN

            (* Create identification string used by debug messages *)
            sID          := CONCAT(CONCAT('[', DWORD_TO_HEXSTR(fbConnect.hSocket.handle, 4, FALSE) ), ']');
            errors.sMessage := CONCAT('CLI.Err', sID);

            IF NOT fbConnect.bError THEN
                IF eState = eSOCKET_CONNECTED THEN(* we are connected *)
                    state := 2;
                END_IF
            ELSE(* connect error: log error *)
                errors.Error(nErrId := fbConnect.nErrId);
            END_IF
        END_IF

    2:(* Data exchange state *)
        bDisconnect := NOT bEnable OR bDisconnect; (* user/internal disconnect requested? *)
        IF bDisconnect AND (tx_state = 0) AND (rx_state = 0) THEN
            state := 3;(* disconnect *)
        ELSE
            (*--------------------------- Send tx data -------------------------------------------*)
            CASE tx_state OF
                0:
                    IF NOT bDisconnect THEN

                        (* forcefully send data each cycle *)

                        (* create the raw datagram *)
                        _byteCount                   := 76;
                        toServer.Header.ByteCount    := HOST_TO_BE32(in := _byteCount);
                        toServer.Header.DatagramType := HOST_TO_BE32(in := MNG_Raw32BitImage);
                        toServer.Header.Counter      := Counter;

                        toServer.Payload[1] := HOST_TO_BE32(18); (* number of signals *)

                        (* BOOL MotorX_00_par1 *)
                        IF Outputs.MotorX_00_par1 THEN
                            toServer.Payload[2] := 16#FFFFFFFF;   (*BOOL *)
                        ELSE
                            toServer.Payload[2] := 0;
                        END_IF;

                        (* BOOL MotorX_00_par2 *)
                        IF Outputs.MotorX_00_par2 THEN
                            toServer.Payload[3] := 16#FFFFFFFF;   (*BOOL *)
                        ELSE
                            toServer.Payload[3] := 0;
                        END_IF;

                        (* FLOAT32 Keksmodul_00_ACT_POS02 *)
                        MEMCPY(destAddr := ADR(DWordBuffer), srcAddr := ADR(Outputs.Keksmodul_00_ACT_POS02), n := 4);
                        toServer.Payload[4] := HOST_TO_BE32(DWordBuffer);

                        (* FLOAT32 Toppingmodul_Bosch_00_ACT_POS02 *)
                        MEMCPY(destAddr := ADR(DWordBuffer), srcAddr := ADR(Outputs.Toppingmodul_Bosch_00_ACT_POS02), n := 4);
                        toServer.Payload[5] := HOST_TO_BE32(DWordBuffer);

                        (* FLOAT32 Toppingmodul_Beckhoff_00_ACT_POS02 *)
                        MEMCPY(destAddr := ADR(DWordBuffer), srcAddr := ADR(Outputs.Toppingmodul_Beckhoff_00_ACT_POS02), n := 4);
                        toServer.Payload[6] := HOST_TO_BE32(DWordBuffer);

                        (* FLOAT32 DosierModul_00_ACT_POS02 *)
                        MEMCPY(destAddr := ADR(DWordBuffer), srcAddr := ADR(Outputs.DosierModul_00_ACT_POS02), n := 4);
                        toServer.Payload[7] := HOST_TO_BE32(DWordBuffer);

                        (* BOOL status_00_on102 *)
                        IF Outputs.status_00_on102 THEN
                            toServer.Payload[8] := 16#FFFFFFFF;   (*BOOL *)
                        ELSE
                            toServer.Payload[8] := 0;
                        END_IF;

                        (* BOOL status_00_on202 *)
                        IF Outputs.status_00_on202 THEN
                            toServer.Payload[9] := 16#FFFFFFFF;   (*BOOL *)
                        ELSE
                            toServer.Payload[9] := 0;
                        END_IF;

                        (* BOOL status_00_on302 *)
                        IF Outputs.status_00_on302 THEN
                            toServer.Payload[10] := 16#FFFFFFFF;   (*BOOL *)
                        ELSE
                            toServer.Payload[10] := 0;
                        END_IF;

                        (* BOOL status_00_on103 *)
                        IF Outputs.status_00_on103 THEN
                            toServer.Payload[11] := 16#FFFFFFFF;   (*BOOL *)
                        ELSE
                            toServer.Payload[11] := 0;
                        END_IF;

                        (* BOOL status_00_on203 *)
                        IF Outputs.status_00_on203 THEN
                            toServer.Payload[12] := 16#FFFFFFFF;   (*BOOL *)
                        ELSE
                            toServer.Payload[12] := 0;
                        END_IF;

                        (* BOOL status_00_on303 *)
                        IF Outputs.status_00_on303 THEN
                            toServer.Payload[13] := 16#FFFFFFFF;   (*BOOL *)
                        ELSE
                            toServer.Payload[13] := 0;
                        END_IF;

                        (* BOOL status_00_on104 *)
                        IF Outputs.status_00_on104 THEN
                            toServer.Payload[14] := 16#FFFFFFFF;   (*BOOL *)
                        ELSE
                            toServer.Payload[14] := 0;
                        END_IF;

                        (* BOOL status_00_on204 *)
                        IF Outputs.status_00_on204 THEN
                            toServer.Payload[15] := 16#FFFFFFFF;   (*BOOL *)
                        ELSE
                            toServer.Payload[15] := 0;
                        END_IF;

                        (* BOOL status_00_on304 *)
                        IF Outputs.status_00_on304 THEN
                            toServer.Payload[16] := 16#FFFFFFFF;   (*BOOL *)
                        ELSE
                            toServer.Payload[16] := 0;
                        END_IF;

                        (* BOOL status_00_on105 *)
                        IF Outputs.status_00_on105 THEN
                            toServer.Payload[17] := 16#FFFFFFFF;   (*BOOL *)
                        ELSE
                            toServer.Payload[17] := 0;
                        END_IF;

                        (* BOOL status_00_on205 *)
                        IF Outputs.status_00_on205 THEN
                            toServer.Payload[18] := 16#FFFFFFFF;   (*BOOL *)
                        ELSE
                            toServer.Payload[18] := 0;
                        END_IF;

                        (* BOOL status_00_on305 *)
                        IF Outputs.status_00_on305 THEN
                            toServer.Payload[19] := 16#FFFFFFFF;   (*BOOL *)
                        ELSE
                            toServer.Payload[19] := 0;
                        END_IF;

                        toServer.Header.SentTime := HOST_TO_BE32(in := clock.systemTime.wMilliseconds + clock.systemTime.wMinute * 60000);

                        (* send frame *)
                        fbSend(bExecute  := FALSE);
                        fbSend(sSrvNetID := '',
                               hSocket   := fbConnect.hSocket,
                               cbLen     := SIZEOF(toServer.Header) + _byteCount,(* size of header + size of user data *)
                               pSrc      := ADR(toServer),(* pointer to the frame data *)
                               bExecute  := TRUE,
                               tTimeout  := T#5s);

                        tx_state := 1;
                    END_IF
                1:(* wait until send not busy *)
                    fbSend( bExecute := FALSE );
                    IF NOT fbSend.bBusy THEN
                        tx_state := 0;
                        IF NOT fbSend.bError THEN(* no error *)
                            ;
                        ELSE(* send error => log error and disconnect *)
                            errors.Error(nErrId := fbSend.nErrId );
                            bDisconnect := TRUE;(* set flag *)
                        END_IF
                    END_IF
            END_CASE

            (* ------------------------------------------- Get/fetch rx data ----------------------------------------------------------------- *)
            CASE rx_state OF
                0:
                    IF NOT bDisconnect THEN
                        pollTimer( IN := TRUE );
                        IF pollTimer.Q THEN
                            pollTimer( IN := FALSE );

                            fbReceive( bExecute := FALSE );
                            fbReceive( 	sSrvNetId	:= '',
                            hSocket		:= fbConnect.hSocket,
                            cbLen		:= SIZEOF(fromServer) - cbReceived,
                            pDest		:= ADR(fromServer) + cbReceived,
                            bExecute	:= TRUE,
                            tTimeout	:= T#5s );
                            rx_state := 1;
                        END_IF
                    END_IF
                1:(* wait until receive not busy *)
                    fbReceive( bExecute := FALSE );
                    IF NOT fbReceive.bBusy THEN
                        rx_state := 0;
                        IF NOT fbReceive.bError THEN
                            IF fbReceive.nRecBytes > 0 THEN (* some bytes received *)

                                pollTimer( PT := T#0s );(* increase polling speed *)
                                cbReceived := cbReceived + fbReceive.nRecBytes;

                                (* parse received bytes *)
                                REPEAT
                                    bAbort := TRUE;(* set flag *)
                                    IF cbReceived >= SIZEOF(fromServer.Header) THEN (* all header bytes received => check header data *)

                                        (* correct header data *)
                                        fromServer.Header.ByteCount    := BE32_TO_HOST(fromServer.Header.ByteCount);
                                        Counter                        := fromServer.Header.Counter;
                                        fromServer.Header.SentTime     := BE32_TO_HOST(fromServer.Header.SentTime);
                                        fromServer.Header.DatagramType := BE32_TO_HOST(fromServer.Header.DatagramType);

                                        IF (fromServer.Header.ByteCount <= SIZEOF( fromServer.Payload))(* check frame (user data) length *)
                                        THEN

                                            cbRx := SIZEOF(fromServer.Header) + fromServer.Header.ByteCount;(* calculate the (expected) length of the rx frame *)
                                            IF cbReceived >= cbRx  THEN (* all frame bytes received? *)

                                               (* currently only use the data on a 32 Bit raw image *)
                                                IF fromServer.Header.DatagramType = MNG_Raw32BitImage THEN

                                                    IF 4 = (fromServer.Header.ByteCount - 4) THEN

                                                        (* BOOL init_sensor_module_x_00_IR *)
                                                        Inputs.init_sensor_module_x_00_IR := fromServer.Payload[2]<>0;

                                                    ELSE(* receive error: invalid frame format/data *)
                                                        errors.Error(nErrId := PLCPRJ_ERROR_INVALID_IO_FORMAT_RECEIVED );
                                                    END_IF

                                                END_IF

                                                MEMMOVE( ADR( fromServer ), ADR( fromServer ) + cbRx,  cbReceived - cbRx );(* shift the remaining rx bytes *)
                                                cbReceived := cbReceived - cbRx;(* recalculate the size of the remaining rx bytes *)

                                                bAbort := FALSE;(* reset flag, try to parse next frame *)

                                                (* ELSE repeat reading *)
                                            END_IF

                                        ELSE(* receive error: invalid frame format/data *)
                                            errors.Error(nErrId := PLCPRJ_ERROR_INVALID_FRAME_FORMAT );
                                            bDisconnect := TRUE;(* set flag *)
                                        END_IF
                                        (* ELSE repeat reading *)
                                    END_IF (* IF cbReceived >= SIZEOF(rxFrame.head) THEN *)

                                UNTIL bAbort
                                END_REPEAT

